LIN {X -0.023,Y -429.187,Z 1281.514,A 0.000,B 0.000,C 90.000,E1 272.465} C_DIS
LIN {X -0.033,Y -422.236,Z 1281.512,A 0.000,B 0.000,C 90.000,E1 272.121} C_DIS
LIN {X -0.038,Y -415.238,Z 1281.510,A 0.000,B 0.000,C 90.000,E1 271.835} C_DIS
LIN {X -0.099,Y -408.071,Z 1281.509,A 0.000,B 0.000,C 90.000,E1 271.604} C_DIS
LIN {X 0.103,Y -401.016,Z 1281.508,A 0.000,B 0.000,C 90.000,E1 271.375} C_DIS
LIN {X 0.112,Y -393.582,Z 1281.507,A 0.000,B 0.000,C 90.000,E1 271.203} C_DIS
LIN {X -0.037,Y -385.526,Z 1281.506,A 0.000,B 0.000,C 90.000,E1 271.088} C_DIS
LIN {X 0.028,Y -376.510,Z 1281.505,A 0.000,B 0.000,C 90.000,E1 270.974} C_DIS
LIN {X -0.122,Y -364.751,Z 1281.505,A 0.000,B 0.000,C 90.000,E1 270.917} C_DIS
LIN {X -0.176,Y -360.433,Z 1281.505,A 0.000,B 0.000,C 90.000,E1 270.917} C_DIS
LIN {X 0.065,Y -181.483,Z 1281.505,A 0.000,B 0.000,C 90.000,E1 270.859} C_DIS
LIN {X 0.085,Y -181.533,Z 1281.499,A 0.000,B 0.000,C 90.000,E1 269.828} C_DIS
LIN {X 0.028,Y -180.907,Z 1281.475,A 0.000,B 0.000,C 90.000,E1 265.469} C_DIS
LIN {X -0.095,Y -180.741,Z 1281.470,A 0.000,B 0.000,C 90.000,E1 264.666} C_DIS
LIN {X 0.006,Y -178.831,Z 1281.442,A 0.000,B 0.000,C 90.000,E1 259.567} C_DIS
LIN {X 0.040,Y -175.875,Z 1281.414,A 0.000,B 0.000,C 90.000,E1 254.464} C_DIS
LIN {X -0.084,Y -173.849,Z 1281.400,A 0.000,B 0.000,C 90.000,E1 251.945} C_DIS
LIN {X 0.070,Y -171.518,Z 1281.380,A 0.000,B 0.000,C 90.000,E1 248.465} C_DIS
LIN {X 0.056,Y -167.744,Z 1281.357,A 0.000,B 0.000,C 90.000,E1 244.152} C_DIS
LIN {X 0.072,Y -166.446,Z 1281.347,A 0.000,B 0.000,C 90.000,E1 242.410} C_DIS
LIN {X -0.016,Y -163.163,Z 1281.328,A 0.000,B 0.000,C 90.000,E1 238.948} C_DIS
LIN {X 0.034,Y -161.121,Z 1281.313,A 0.000,B 0.000,C 90.000,E1 236.294} C_DIS
LIN {X -0.063,Y -157.144,Z 1281.288,A 0.000,B 0.000,C 90.000,E1 231.904} C_DIS
LIN {X -0.040,Y -155.877,Z 1281.278,A 0.000,B 0.000,C 90.000,E1 230.114} C_DIS
LIN {X -0.081,Y -152.127,Z 1281.253,A 0.000,B 0.000,C 90.000,E1 225.648} C_DIS
LIN {X -0.060,Y -150.377,Z 1281.238,A 0.000,B 0.000,C 90.000,E1 222.933} C_DIS
LIN {X -0.035,Y -147.110,Z 1281.213,A 0.000,B 0.000,C 90.000,E1 218.382} C_DIS
LIN {X -0.044,Y -145.676,Z 1281.198,A 0.000,B 0.000,C 90.000,E1 215.644} C_DIS
LIN {X -0.046,Y -143.059,Z 1281.172,A 0.000,B 0.000,C 90.000,E1 211.052} C_DIS
LIN {X 0.012,Y -141.681,Z 1281.152,A 0.000,B 0.000,C 90.000,E1 207.334} C_DIS
LIN {X -0.010,Y -139.457,Z 1281.116,A 0.000,B 0.000,C 90.000,E1 200.844} C_DIS
LIN {X 0.040,Y -139.191,Z 1281.105,A 0.000,B 0.000,C 90.000,E1 198.960} C_DIS
LIN {X 0.064,Y -138.324,Z 1281.054,A 0.000,B 0.000,C 90.000,E1 189.613} C_DIS
LIN {X -0.068,Y -139.455,Z 1281.007,A 0.000,B 0.000,C 90.000,E1 181.260} C_DIS
LIN {X 0.012,Y -141.005,Z 1280.976,A 0.000,B 0.000,C 90.000,E1 175.641} C_DIS
LIN {X -0.039,Y -142.759,Z 1280.955,A 0.000,B 0.000,C 90.000,E1 171.951} C_DIS
LIN {X 0.058,Y -145.164,Z 1280.930,A 0.000,B 0.000,C 90.000,E1 167.297} C_DIS
LIN {X 0.050,Y -147.786,Z 1280.909,A 0.000,B 0.000,C 90.000,E1 163.630} C_DIS
LIN {X -0.012,Y -150.466,Z 1280.889,A 0.000,B 0.000,C 90.000,E1 160.007} C_DIS
LIN {X 0.062,Y -153.918,Z 1280.869,A 0.000,B 0.000,C 90.000,E1 156.357} C_DIS
LIN {X -0.013,Y -157.329,Z 1280.849,A 0.000,B 0.000,C 90.000,E1 152.794} C_DIS
LIN {X 0.071,Y -161.519,Z 1280.829,A 0.000,B 0.000,C 90.000,E1 149.203} C_DIS
LIN {X -0.053,Y -165.718,Z 1280.809,A 0.000,B 0.000,C 90.000,E1 145.722} C_DIS
LIN {X 0.072,Y -170.666,Z 1280.790,A 0.000,B 0.000,C 90.000,E1 142.190} C_DIS
LIN {X -0.015,Y -175.541,Z 1280.771,A 0.000,B 0.000,C 90.000,E1 138.771} C_DIS
LIN {X -0.022,Y -181.160,Z 1280.752,A 0.000,B 0.000,C 90.000,E1 135.364} C_DIS
LIN {X -0.025,Y -186.614,Z 1280.733,A 0.000,B 0.000,C 90.000,E1 132.000} C_DIS
LIN {X 0.046,Y -191.223,Z 1280.719,A 0.000,B 0.000,C 90.000,E1 129.483} C_DIS
LIN {X -0.032,Y -197.039,Z 1280.701,A 0.000,B 0.000,C 90.000,E1 126.217} C_DIS
LIN {X -0.072,Y -199.854,Z 1280.693,A 0.000,B 0.000,C 90.000,E1 124.818} C_DIS
LIN {X -0.149,Y -309.309,Z 1280.693,A 0.000,B 0.000,C 90.000,E1 124.818} C_DIS
LIN {X -0.180,Y -315.387,Z 1280.692,A 0.000,B 0.000,C 90.000,E1 124.612} C_DIS
LIN {X 0.081,Y -318.330,Z 1280.691,A 0.000,B 0.000,C 90.000,E1 124.326} C_DIS
LIN {X 0.009,Y -322.051,Z 1280.688,A 0.000,B 0.000,C 90.000,E1 123.865} C_DIS
LIN {X -0.184,Y -323.801,Z 1280.686,A 0.000,B 0.000,C 90.000,E1 123.579} C_DIS
LIN {X 0.070,Y -325.164,Z 1280.685,A 0.000,B 0.000,C 90.000,E1 123.214} C_DIS
LIN {X 0.002,Y -336.874,Z 1280.667,A 0.000,B 0.000,C 90.000,E1 120.079} C_DIS
LIN {X -0.030,Y -348.823,Z 1280.652,A 0.000,B 0.000,C 90.000,E1 117.308} C_DIS
LIN {X -0.055,Y -362.234,Z 1280.637,A 0.000,B 0.000,C 90.000,E1 114.591} C_DIS
LIN {X 0.061,Y -375.474,Z 1280.623,A 0.000,B 0.000,C 90.000,E1 112.206} C_DIS
LIN {X 0.091,Y -390.050,Z 1280.611,A 0.000,B 0.000,C 90.000,E1 109.885} C_DIS
LIN {X -0.017,Y -406.067,Z 1280.598,A 0.000,B 0.000,C 90.000,E1 107.638} C_DIS
LIN {X 0.015,Y -423.637,Z 1280.586,A 0.000,B 0.000,C 90.000,E1 105.426} C_DIS
LIN {X -0.129,Y -442.844,Z 1280.574,A 0.000,B 0.000,C 90.000,E1 103.300} C_DIS
LIN {X -0.134,Y -462.963,Z 1280.563,A 0.000,B 0.000,C 90.000,E1 101.299} C_DIS
LIN {X -0.203,Y -475.789,Z 1280.556,A 0.000,B 0.000,C 90.000,E1 100.141} C_DIS
LIN {X -0.134,Y -477.907,Z 1280.555,A 0.000,B 0.000,C 90.000,E1 99.905} C_DIS
LIN {X 0.209,Y -479.663,Z 1280.554,A 0.000,B 0.000,C 90.000,E1 99.613} C_DIS
LIN {X 0.077,Y -480.981,Z 1280.552,A 0.000,B 0.000,C 90.000,E1 99.378} C_DIS
LIN {X 0.233,Y -482.621,Z 1280.549,A 0.000,B 0.000,C 90.000,E1 98.859} C_DIS
LIN {X -0.078,Y -483.190,Z 1280.547,A 0.000,B 0.000,C 90.000,E1 98.398} C_DIS
LIN {X 0.166,Y -482.782,Z 1280.544,A 0.000,B 0.000,C 90.000,E1 97.871} C_DIS
LIN {X -0.133,Y -481.337,Z 1280.541,A 0.000,B 0.000,C 90.000,E1 97.409} C_DIS
LIN {X 0.164,Y -480.150,Z 1280.540,A 0.000,B 0.000,C 90.000,E1 97.125} C_DIS
LIN {X 0.043,Y -478.567,Z 1280.538,A 0.000,B 0.000,C 90.000,E1 96.891} C_DIS
LIN {X 0.044,Y -463.775,Z 1280.527,A 0.000,B 0.000,C 90.000,E1 94.878} C_DIS
LIN {X 0.139,Y -446.409,Z 1280.513,A 0.000,B 0.000,C 90.000,E1 92.293} C_DIS
LIN {X -0.012,Y -431.889,Z 1280.500,A 0.000,B 0.000,C 90.000,E1 89.943} C_DIS
LIN {X 0.013,Y -417.151,Z 1280.485,A 0.000,B 0.000,C 90.000,E1 87.249} C_DIS
LIN {X -0.060,Y -405.581,Z 1280.473,A 0.000,B 0.000,C 90.000,E1 85.065} C_DIS
LIN {X -0.059,Y -396.894,Z 1280.463,A 0.000,B 0.000,C 90.000,E1 83.394} C_DIS
LIN {X -0.166,Y -386.549,Z 1280.452,A 0.000,B 0.000,C 90.000,E1 81.432} C_DIS
LIN {X -0.022,Y -377.434,Z 1280.443,A 0.000,B 0.000,C 90.000,E1 79.690} C_DIS
LIN {X 0.022,Y -367.963,Z 1280.433,A 0.000,B 0.000,C 90.000,E1 77.937} C_DIS
LIN {X -0.027,Y -358.150,Z 1280.423,A 0.000,B 0.000,C 90.000,E1 76.172} C_DIS
LIN {X 0.097,Y -346.573,Z 1280.411,A 0.000,B 0.000,C 90.000,E1 74.047} C_DIS
LIN {X -0.162,Y -335.085,Z 1280.400,A 0.000,B 0.000,C 90.000,E1 71.945} C_DIS
LIN {X 0.088,Y -320.715,Z 1280.384,A 0.000,B 0.000,C 90.000,E1 69.082} C_DIS
LIN {X 0.105,Y -304.373,Z 1280.364,A 0.000,B 0.000,C 90.000,E1 65.537} C_DIS
LIN {X -0.024,Y -293.664,Z 1280.349,A 0.000,B 0.000,C 90.000,E1 62.922} C_DIS
LIN {X 0.112,Y -284.252,Z 1280.335,A 0.000,B 0.000,C 90.000,E1 60.205} C_DIS
LIN {X -0.136,Y -273.724,Z 1280.316,A 0.000,B 0.000,C 90.000,E1 56.834} C_DIS
LIN {X -0.077,Y -264.169,Z 1280.296,A 0.000,B 0.000,C 90.000,E1 53.336} C_DIS
LIN {X 0.018,Y -256.937,Z 1280.281,A 0.000,B 0.000,C 90.000,E1 50.481} C_DIS
LIN {X -0.105,Y -249.955,Z 1280.265,A 0.000,B 0.000,C 90.000,E1 47.634} C_DIS
LIN {X 0.057,Y -241.694,Z 1280.244,A 0.000,B 0.000,C 90.000,E1 43.947} C_DIS
LIN {X -0.012,Y -233.958,Z 1280.224,A 0.000,B 0.000,C 90.000,E1 40.253} C_DIS
LIN {X -0.080,Y -227.073,Z 1280.203,A 0.000,B 0.000,C 90.000,E1 36.503} C_DIS
LIN {X -0.041,Y -220.916,Z 1280.182,A 0.000,B 0.000,C 90.000,E1 32.673} C_DIS
LIN {X -0.103,Y -215.433,Z 1280.160,A 0.000,B 0.000,C 90.000,E1 28.821} C_DIS
LIN {X -0.068,Y -210.589,Z 1280.138,A 0.000,B 0.000,C 90.000,E1 24.899} C_DIS
LIN {X 0.046,Y -205.645,Z 1280.112,A 0.000,B 0.000,C 90.000,E1 20.120} C_DIS
LIN {X 0.072,Y -201.484,Z 1280.085,A 0.000,B 0.000,C 90.000,E1 15.315} C_DIS
LIN {X 0.062,Y -197.828,Z 1280.054,A 0.000,B 0.000,C 90.000,E1 9.670} C_DIS
LIN {X 0.062,Y -195.327,Z 1280.013,A 0.000,B 0.000,C 90.000,E1 2.350} C_DIS
LIN {X 0.014,Y -196.745,Z 1279.957,A 0.000,B 0.000,C 90.000,E1 352.186} C_DIS
LIN {X -0.045,Y -200.083,Z 1279.925,A 0.000,B 0.000,C 90.000,E1 346.520} C_DIS
LIN {X -0.067,Y -204.142,Z 1279.898,A 0.000,B 0.000,C 90.000,E1 341.692} C_DIS
LIN {X 0.045,Y -208.261,Z 1279.876,A 0.000,B 0.000,C 90.000,E1 337.667} C_DIS
LIN {X 0.020,Y -213.164,Z 1279.854,A 0.000,B 0.000,C 90.000,E1 333.717} C_DIS
LIN {X 0.055,Y -218.767,Z 1279.832,A 0.000,B 0.000,C 90.000,E1 329.793} C_DIS
LIN {X 0.047,Y -225.145,Z 1279.811,A 0.000,B 0.000,C 90.000,E1 325.928} C_DIS
LIN {X 0.065,Y -232.457,Z 1279.790,A 0.000,B 0.000,C 90.000,E1 322.110} C_DIS
LIN {X 0.016,Y -240.603,Z 1279.769,A 0.000,B 0.000,C 90.000,E1 318.366} C_DIS
LIN {X 0.016,Y -248.933,Z 1279.750,A 0.000,B 0.000,C 90.000,E1 315.040} C_DIS
LIN {X 0.065,Y -257.259,Z 1279.734,A 0.000,B 0.000,C 90.000,E1 312.123} C_DIS
LIN {X -0.089,Y -264.405,Z 1279.722,A 0.000,B 0.000,C 90.000,E1 310.011} C_DIS
LIN {X 0.019,Y -271.052,Z 1279.712,A 0.000,B 0.000,C 90.000,E1 308.222} C_DIS
LIN {X -0.001,Y -279.977,Z 1279.701,A 0.000,B 0.000,C 90.000,E1 306.137} C_DIS
LIN {X 0.059,Y -289.953,Z 1279.689,A 0.000,B 0.000,C 90.000,E1 304.072} C_DIS
LIN {X -0.085,Y -301.013,Z 1279.678,A 0.000,B 0.000,C 90.000,E1 302.084} C_DIS
LIN {X 0.038,Y -311.291,Z 1279.669,A 0.000,B 0.000,C 90.000,E1 300.413} C_DIS
LIN {X 0.059,Y -327.603,Z 1279.656,A 0.000,B 0.000,C 90.000,E1 298.153} C_DIS
LIN {X -0.025,Y -347.797,Z 1279.643,A 0.000,B 0.000,C 90.000,E1 295.668} C_DIS
LIN {X 0.113,Y -360.704,Z 1279.634,A 0.000,B 0.000,C 90.000,E1 294.155} C_DIS
LIN {X -0.040,Y -373.638,Z 1279.626,A 0.000,B 0.000,C 90.000,E1 292.695} C_DIS
LIN {X -0.144,Y -386.003,Z 1279.618,A 0.000,B 0.000,C 90.000,E1 291.280} C_DIS
LIN {X 0.233,Y -410.888,Z 1279.603,A 0.000,B 0.000,C 90.000,E1 288.417} C_DIS
LIN {X 0.117,Y -420.946,Z 1279.596,A 0.000,B 0.000,C 90.000,E1 287.347} C_DIS
LIN {X 0.132,Y -430.448,Z 1279.590,A 0.000,B 0.000,C 90.000,E1 286.260} C_DIS
LIN {X -0.066,Y -437.039,Z 1279.586,A 0.000,B 0.000,C 90.000,E1 285.481} C_DIS
LIN {X 0.109,Y -443.024,Z 1279.582,A 0.000,B 0.000,C 90.000,E1 284.662} C_DIS
LIN {X 0.017,Y -448.346,Z 1279.577,A 0.000,B 0.000,C 90.000,E1 283.883} C_DIS
LIN {X -0.136,Y -452.992,Z 1279.573,A 0.000,B 0.000,C 90.000,E1 283.119} C_DIS
LIN {X 0.193,Y -456.947,Z 1279.568,A 0.000,B 0.000,C 90.000,E1 282.299} C_DIS
LIN {X -0.162,Y -459.237,Z 1279.566,A 0.000,B 0.000,C 90.000,E1 281.827} C_DIS
LIN {X -0.056,Y -461.228,Z 1279.563,A 0.000,B 0.000,C 90.000,E1 281.299} C_DIS
LIN {X -0.031,Y -462.946,Z 1279.560,A 0.000,B 0.000,C 90.000,E1 280.782} C_DIS
LIN {X 0.094,Y -464.342,Z 1279.557,A 0.000,B 0.000,C 90.000,E1 280.254} C_DIS
LIN {X 0.226,Y -465.390,Z 1279.554,A 0.000,B 0.000,C 90.000,E1 279.726} C_DIS
LIN {X -0.171,Y -466.115,Z 1279.551,A 0.000,B 0.000,C 90.000,E1 279.265} C_DIS
LIN {X -0.099,Y -466.471,Z 1279.548,A 0.000,B 0.000,C 90.000,E1 278.746} C_DIS
LIN {X 0.046,Y -466.382,Z 1279.546,A 0.000,B 0.000,C 90.000,E1 278.219} C_DIS
LIN {X 0.125,Y -465.867,Z 1279.543,A 0.000,B 0.000,C 90.000,E1 277.701} C_DIS
LIN {X 0.205,Y -464.875,Z 1279.540,A 0.000,B 0.000,C 90.000,E1 277.182} C_DIS
LIN {X -0.178,Y -463.420,Z 1279.537,A 0.000,B 0.000,C 90.000,E1 276.720} C_DIS
LIN {X -0.105,Y -461.545,Z 1279.534,A 0.000,B 0.000,C 90.000,E1 276.201} C_DIS
LIN {X 0.231,Y -458.114,Z 1279.530,A 0.000,B 0.000,C 90.000,E1 275.391} C_DIS
LIN {X -0.227,Y -455.355,Z 1279.527,A 0.000,B 0.000,C 90.000,E1 274.935} C_DIS
LIN {X -0.203,Y -452.069,Z 1279.524,A 0.000,B 0.000,C 90.000,E1 274.416} C_DIS
LIN {X -0.198,Y -447.836,Z 1279.521,A 0.000,B 0.000,C 90.000,E1 273.898} C_DIS
LIN {X 0.007,Y -445.358,Z 1279.520,A 0.000,B 0.000,C 90.000,E1 273.612} C_DIS
LIN {X -0.003,Y -439.433,Z 1279.517,A 0.000,B 0.000,C 90.000,E1 273.094} C_DIS
LIN {X 0.067,Y -432.981,Z 1279.515,A 0.000,B 0.000,C 90.000,E1 272.636} C_DIS
LIN {X 0.187,Y -426.045,Z 1279.513,A 0.000,B 0.000,C 90.000,E1 272.236} C_DIS
LIN {X -0.035,Y -419.065,Z 1279.511,A 0.000,B 0.000,C 90.000,E1 271.949} C_DIS
LIN {X 0.193,Y -412.131,Z 1279.509,A 0.000,B 0.000,C 90.000,E1 271.661} C_DIS
LIN {X -0.145,Y -405.059,Z 1279.508,A 0.000,B 0.000,C 90.000,E1 271.489} C_DIS
LIN {X 0.141,Y -397.896,Z 1279.507,A 0.000,B 0.000,C 90.000,E1 271.260} C_DIS
LIN {X -0.184,Y -389.490,Z 1279.506,A 0.000,B 0.000,C 90.000,E1 271.146} C_DIS
LIN {X 0.174,Y -381.137,Z 1279.506,A 0.000,B 0.000,C 90.000,E1 270.974} C_DIS
LIN {X -0.073,Y -370.345,Z 1279.505,A 0.000,B 0.000,C 90.000,E1 270.917} C_DIS
LIN {X 0.010,Y -359.049,Z 1279.505,A 0.000,B 0.000,C 90.000,E1 270.859} C_DIS
LIN {X -0.023,Y -181.490,Z 1279.505,A 0.000,B 0.000,C 90.000,E1 270.859} C_DIS
LIN {X -0.002,Y -181.525,Z 1279.499,A 0.000,B 0.000,C 90.000,E1 269.828} C_DIS
LIN {X -0.059,Y -180.907,Z 1279.475,A 0.000,B 0.000,C 90.000,E1 265.469} C_DIS
LIN {X -0.003,Y -180.728,Z 1279.470,A 0.000,B 0.000,C 90.000,E1 264.609} C_DIS
LIN {X 0.095,Y -178.817,Z 1279.442,A 0.000,B 0.000,C 90.000,E1 259.511} C_DIS
LIN {X 0.001,Y -175.861,Z 1279.414,A 0.000,B 0.000,C 90.000,E1 254.448} C_DIS
LIN {X 0.050,Y -173.827,Z 1279.399,A 0.000,B 0.000,C 90.000,E1 251.873} C_DIS
LIN {X -0.014,Y -171.495,Z 1279.380,A 0.000,B 0.000,C 90.000,E1 248.465} C_DIS
LIN {X -0.028,Y -167.724,Z 1279.356,A 0.000,B 0.000,C 90.000,E1 244.152} C_DIS
LIN {X -0.012,Y -166.417,Z 1279.347,A 0.000,B 0.000,C 90.000,E1 242.410} C_DIS
LIN {X -0.013,Y -163.140,Z 1279.327,A 0.000,B 0.000,C 90.000,E1 238.918} C_DIS
LIN {X -0.048,Y -161.093,Z 1279.313,A 0.000,B 0.000,C 90.000,E1 236.294} C_DIS
LIN {X -0.064,Y -157.822,Z 1279.293,A 0.000,B 0.000,C 90.000,E1 232.763} C_DIS
LIN {X 0.000,Y -155.856,Z 1279.278,A 0.000,B 0.000,C 90.000,E1 230.070} C_DIS
LIN {X 0.055,Y -152.105,Z 1279.253,A 0.000,B 0.000,C 90.000,E1 225.567} C_DIS
LIN {X 0.074,Y -150.356,Z 1279.238,A 0.000,B 0.000,C 90.000,E1 222.852} C_DIS
LIN {X 0.002,Y -147.092,Z 1279.213,A 0.000,B 0.000,C 90.000,E1 218.338} C_DIS
LIN {X -0.003,Y -145.663,Z 1279.198,A 0.000,B 0.000,C 90.000,E1 215.598} C_DIS
LIN {X 0.001,Y -143.045,Z 1279.172,A 0.000,B 0.000,C 90.000,E1 211.003} C_DIS
LIN {X 0.001,Y -141.669,Z 1279.152,A 0.000,B 0.000,C 90.000,E1 207.308} C_DIS
LIN {X 0.046,Y -139.451,Z 1279.116,A 0.000,B 0.000,C 90.000,E1 200.791} C_DIS
LIN {X -0.034,Y -139.186,Z 1279.105,A 0.000,B 0.000,C 90.000,E1 198.960} C_DIS
LIN {X -0.011,Y -138.321,Z 1279.053,A 0.000,B 0.000,C 90.000,E1 189.613} C_DIS
LIN {X -0.003,Y -139.461,Z 1279.007,A 0.000,B 0.000,C 90.000,E1 181.203} C_DIS
LIN {X -0.064,Y -141.018,Z 1278.976,A 0.000,B 0.000,C 90.000,E1 175.641} C_DIS
LIN {X 0.027,Y -142.772,Z 1278.955,A 0.000,B 0.000,C 90.000,E1 171.894} C_DIS
LIN {X 0.013,Y -145.184,Z 1278.929,A 0.000,B 0.000,C 90.000,E1 167.285} C_DIS
LIN {X 0.015,Y -147.805,Z 1278.909,A 0.000,B 0.000,C 90.000,E1 163.614} C_DIS
LIN {X -0.091,Y -150.491,Z 1278.889,A 0.000,B 0.000,C 90.000,E1 160.007} C_DIS
LIN {X -0.018,Y -153.949,Z 1278.869,A 0.000,B 0.000,C 90.000,E1 156.357} C_DIS
LIN {X 0.045,Y -157.359,Z 1278.849,A 0.000,B 0.000,C 90.000,E1 152.743} C_DIS
LIN {X -0.011,Y -161.557,Z 1278.829,A 0.000,B 0.000,C 90.000,E1 149.203} C_DIS
LIN {X 0.000,Y -165.755,Z 1278.809,A 0.000,B 0.000,C 90.000,E1 145.674} C_DIS
LIN {X -0.013,Y -170.710,Z 1278.790,A 0.000,B 0.000,C 90.000,E1 142.190} C_DIS
LIN {X 0.031,Y -175.583,Z 1278.771,A 0.000,B 0.000,C 90.000,E1 138.728} C_DIS
LIN {X 0.018,Y -181.201,Z 1278.752,A 0.000,B 0.000,C 90.000,E1 135.324} C_DIS
LIN {X 0.011,Y -186.663,Z 1278.733,A 0.000,B 0.000,C 90.000,E1 131.962} C_DIS
LIN {X -0.045,Y -191.268,Z 1278.719,A 0.000,B 0.000,C 90.000,E1 129.483} C_DIS
LIN {X 0.035,Y -197.090,Z 1278.701,A 0.000,B 0.000,C 90.000,E1 126.171} C_DIS
LIN {X -0.115,Y -199.881,Z 1278.693,A 0.000,B 0.000,C 90.000,E1 124.818} C_DIS
LIN {X 0.039,Y -309.317,Z 1278.693,A 0.000,B 0.000,C 90.000,E1 124.771} C_DIS
LIN {X 0.104,Y -310.853,Z 1278.693,A 0.000,B 0.000,C 90.000,E1 124.739} C_DIS
LIN {X 0.112,Y -315.626,Z 1278.692,A 0.000,B 0.000,C 90.000,E1 124.532} C_DIS
LIN {X 0.034,Y -318.780,Z 1278.690,A 0.000,B 0.000,C 90.000,E1 124.278} C_DIS
LIN {X 0.040,Y -322.447,Z 1278.688,A 0.000,B 0.000,C 90.000,E1 123.785} C_DIS
LIN {X -0.153,Y -324.111,Z 1278.686,A 0.000,B 0.000,C 90.000,E1 123.499} C_DIS
LIN {X 0.021,Y -326.513,Z 1278.682,A 0.000,B 0.000,C 90.000,E1 122.832} C_DIS
LIN {X 0.038,Y -337.143,Z 1278.667,A 0.000,B 0.000,C 90.000,E1 120.001} C_DIS
LIN {X -0.152,Y -349.128,Z 1278.651,A 0.000,B 0.000,C 90.000,E1 117.257} C_DIS
LIN {X -0.015,Y -362.578,Z 1278.636,A 0.000,B 0.000,C 90.000,E1 114.515} C_DIS
LIN {X -0.038,Y -375.854,Z 1278.623,A 0.000,B 0.000,C 90.000,E1 112.153} C_DIS
LIN {X 0.136,Y -390.471,Z 1278.610,A 0.000,B 0.000,C 90.000,E1 109.812} C_DIS
LIN {X -0.092,Y -406.531,Z 1278.598,A 0.000,B 0.000,C 90.000,E1 107.583} C_DIS
LIN {X -0.047,Y -424.147,Z 1278.585,A 0.000,B 0.000,C 90.000,E1 105.371} C_DIS
LIN {X -0.170,Y -443.398,Z 1278.573,A 0.000,B 0.000,C 90.000,E1 103.244} C_DIS
LIN {X -0.135,Y -463.534,Z 1278.562,A 0.000,B 0.000,C 90.000,E1 101.243} C_DIS
LIN {X -0.095,Y -476.300,Z 1278.556,A 0.000,B 0.000,C 90.000,E1 100.074} C_DIS
LIN {X -0.103,Y -478.251,Z 1278.555,A 0.000,B 0.000,C 90.000,E1 99.849} C_DIS
LIN {X -0.233,Y -479.885,Z 1278.553,A 0.000,B 0.000,C 90.000,E1 99.613} C_DIS
LIN {X 0.111,Y -481.109,Z 1278.552,A 0.000,B 0.000,C 90.000,E1 99.321} C_DIS
LIN {X -0.208,Y -482.606,Z 1278.549,A 0.000,B 0.000,C 90.000,E1 98.859} C_DIS
LIN {X -0.041,Y -483.053,Z 1278.546,A 0.000,B 0.000,C 90.000,E1 98.341} C_DIS
LIN {X 0.203,Y -482.525,Z 1278.544,A 0.000,B 0.000,C 90.000,E1 97.814} C_DIS
LIN {X -0.096,Y -480.940,Z 1278.541,A 0.000,B 0.000,C 90.000,E1 97.352} C_DIS
LIN {X 0.200,Y -479.664,Z 1278.539,A 0.000,B 0.000,C 90.000,E1 97.068} C_DIS
LIN {X -0.105,Y -476.050,Z 1278.537,A 0.000,B 0.000,C 90.000,E1 96.606} C_DIS
LIN {X 0.187,Y -456.152,Z 1278.521,A 0.000,B 0.000,C 90.000,E1 93.784} C_DIS
LIN {X 0.202,Y -437.608,Z 1278.505,A 0.000,B 0.000,C 90.000,E1 90.917} C_DIS
LIN {X 0.085,Y -420.993,Z 1278.489,A 0.000,B 0.000,C 90.000,E1 87.993} C_DIS
LIN {X -0.032,Y -410.826,Z 1278.478,A 0.000,B 0.000,C 90.000,E1 86.102} C_DIS
LIN {X 0.104,Y -400.755,Z 1278.468,A 0.000,B 0.000,C 90.000,E1 84.147} C_DIS
LIN {X 0.059,Y -391.959,Z 1278.458,A 0.000,B 0.000,C 90.000,E1 82.470} C_DIS
LIN {X -0.135,Y -383.032,Z 1278.449,A 0.000,B 0.000,C 90.000,E1 80.792} C_DIS
LIN {X -0.055,Y -373.799,Z 1278.439,A 0.000,B 0.000,C 90.000,E1 79.050} C_DIS
LIN {X 0.001,Y -364.189,Z 1278.429,A 0.000,B 0.000,C 90.000,E1 77.285} C_DIS
LIN {X -0.111,Y -354.302,Z 1278.419,A 0.000,B 0.000,C 90.000,E1 75.519} C_DIS
LIN {X 0.030,Y -342.736,Z 1278.408,A 0.000,B 0.000,C 90.000,E1 73.378} C_DIS
LIN {X 0.018,Y -331.311,Z 1278.396,A 0.000,B 0.000,C 90.000,E1 71.221} C_DIS
LIN {X -0.142,Y -317.169,Z 1278.380,A 0.000,B 0.000,C 90.000,E1 68.411} C_DIS
LIN {X -0.010,Y -302.578,Z 1278.362,A 0.000,B 0.000,C 90.000,E1 65.153} C_DIS
LIN {X 0.089,Y -293.315,Z 1278.349,A 0.000,B 0.000,C 90.000,E1 62.820} C_DIS
LIN {X 0.067,Y -282.815,Z 1278.332,A 0.000,B 0.000,C 90.000,E1 59.793} C_DIS
LIN {X 0.105,Y -271.391,Z 1278.311,A 0.000,B 0.000,C 90.000,E1 56.008} C_DIS
LIN {X -0.132,Y -261.948,Z 1278.292,A 0.000,B 0.000,C 90.000,E1 52.557} C_DIS
LIN {X 0.067,Y -254.786,Z 1278.276,A 0.000,B 0.000,C 90.000,E1 49.666} C_DIS
LIN {X 0.051,Y -247.863,Z 1278.260,A 0.000,B 0.000,C 90.000,E1 46.782} C_DIS
LIN {X -0.031,Y -239.732,Z 1278.240,A 0.000,B 0.000,C 90.000,E1 43.137} C_DIS
LIN {X 0.011,Y -232.146,Z 1278.219,A 0.000,B 0.000,C 90.000,E1 39.402} C_DIS
LIN {X 0.103,Y -225.408,Z 1278.198,A 0.000,B 0.000,C 90.000,E1 35.598} C_DIS
LIN {X -0.033,Y -219.368,Z 1278.177,A 0.000,B 0.000,C 90.000,E1 31.799} C_DIS
LIN {X 0.044,Y -213.971,Z 1278.155,A 0.000,B 0.000,C 90.000,E1 27.897} C_DIS
LIN {X -0.044,Y -208.360,Z 1278.129,A 0.000,B 0.000,C 90.000,E1 23.206} C_DIS
LIN {X 0.030,Y -204.388,Z 1278.107,A 0.000,B 0.000,C 90.000,E1 19.214} C_DIS
LIN {X 0.006,Y -200.386,Z 1278.080,A 0.000,B 0.000,C 90.000,E1 14.411} C_DIS
LIN {X 0.021,Y -197.007,Z 1278.049,A 0.000,B 0.000,C 90.000,E1 8.746} C_DIS
LIN {X 0.000,Y -194.842,Z 1278.000,A 0.000,B 0.000,C 90.000,E1 360.000} C_DIS
LIN {X -0.015,Y -196.955,Z 1277.952,A 0.000,B 0.000,C 90.000,E1 351.376} C_DIS
LIN {X -0.025,Y -200.598,Z 1277.921,A 0.000,B 0.000,C 90.000,E1 345.700} C_DIS
LIN {X 0.022,Y -204.837,Z 1277.894,A 0.000,B 0.000,C 90.000,E1 340.859} C_DIS
LIN {X 0.029,Y -209.163,Z 1277.872,A 0.000,B 0.000,C 90.000,E1 336.869} C_DIS
LIN {X 0.021,Y -214.204,Z 1277.850,A 0.000,B 0.000,C 90.000,E1 332.922} C_DIS
LIN {X 0.097,Y -219.966,Z 1277.828,A 0.000,B 0.000,C 90.000,E1 328.997} C_DIS
LIN {X -0.066,Y -226.542,Z 1277.807,A 0.000,B 0.000,C 90.000,E1 325.182} C_DIS
LIN {X -0.057,Y -234.041,Z 1277.785,A 0.000,B 0.000,C 90.000,E1 321.376} C_DIS
LIN {X -0.065,Y -242.379,Z 1277.765,A 0.000,B 0.000,C 90.000,E1 317.634} C_DIS
LIN {X -0.031,Y -251.916,Z 1277.744,A 0.000,B 0.000,C 90.000,E1 313.947} C_DIS
LIN {X 0.095,Y -259.526,Z 1277.730,A 0.000,B 0.000,C 90.000,E1 311.391} C_DIS
LIN {X -0.010,Y -266.950,Z 1277.718,A 0.000,B 0.000,C 90.000,E1 309.277} C_DIS
LIN {X -0.027,Y -273.884,Z 1277.708,A 0.000,B 0.000,C 90.000,E1 307.523} C_DIS
LIN {X 0.011,Y -283.153,Z 1277.697,A 0.000,B 0.000,C 90.000,E1 305.438} C_DIS
LIN {X 0.137,Y -293.485,Z 1277.686,A 0.000,B 0.000,C 90.000,E1 303.372} C_DIS
LIN {X 0.044,Y -302.915,Z 1277.676,A 0.000,B 0.000,C 90.000,E1 301.720} C_DIS
LIN {X -0.008,Y -311.200,Z 1277.669,A 0.000,B 0.000,C 90.000,E1 300.413} C_DIS
LIN {X 0.008,Y -327.553,Z 1277.656,A 0.000,B 0.000,C 90.000,E1 298.153} C_DIS
LIN {X -0.064,Y -347.717,Z 1277.643,A 0.000,B 0.000,C 90.000,E1 295.668} C_DIS
LIN {X 0.060,Y -360.651,Z 1277.634,A 0.000,B 0.000,C 90.000,E1 294.155} C_DIS
LIN {X -0.094,Y -373.586,Z 1277.626,A 0.000,B 0.000,C 90.000,E1 292.695} C_DIS
LIN {X -0.016,Y -386.211,Z 1277.618,A 0.000,B 0.000,C 90.000,E1 291.227} C_DIS
LIN {X 0.208,Y -410.901,Z 1277.602,A 0.000,B 0.000,C 90.000,E1 288.417} C_DIS
LIN {X 0.109,Y -420.945,Z 1277.596,A 0.000,B 0.000,C 90.000,E1 287.347} C_DIS
LIN {X 0.132,Y -430.438,Z 1277.590,A 0.000,B 0.000,C 90.000,E1 286.260} C_DIS
LIN {X -0.066,Y -437.049,Z 1277.586,A 0.000,B 0.000,C 90.000,E1 285.481} C_DIS
LIN {X 0.108,Y -443.037,Z 1277.582,A 0.000,B 0.000,C 90.000,E1 284.662} C_DIS
LIN {X 0.015,Y -448.361,Z 1277.577,A 0.000,B 0.000,C 90.000,E1 283.883} C_DIS
LIN {X -0.137,Y -453.036,Z 1277.573,A 0.000,B 0.000,C 90.000,E1 283.119} C_DIS
LIN {X 0.192,Y -456.997,Z 1277.568,A 0.000,B 0.000,C 90.000,E1 282.299} C_DIS
LIN {X -0.162,Y -459.281,Z 1277.566,A 0.000,B 0.000,C 90.000,E1 281.827} C_DIS
LIN {X -0.056,Y -461.252,Z 1277.563,A 0.000,B 0.000,C 90.000,E1 281.299} C_DIS
LIN {X -0.031,Y -462.980,Z 1277.560,A 0.000,B 0.000,C 90.000,E1 280.782} C_DIS
LIN {X 0.094,Y -464.363,Z 1277.557,A 0.000,B 0.000,C 90.000,E1 280.254} C_DIS
LIN {X 0.227,Y -465.437,Z 1277.554,A 0.000,B 0.000,C 90.000,E1 279.726} C_DIS
LIN {X -0.170,Y -466.189,Z 1277.551,A 0.000,B 0.000,C 90.000,E1 279.265} C_DIS
LIN {X -0.099,Y -466.527,Z 1277.548,A 0.000,B 0.000,C 90.000,E1 278.746} C_DIS
LIN {X 0.047,Y -466.474,Z 1277.546,A 0.000,B 0.000,C 90.000,E1 278.219} C_DIS
LIN {X 0.127,Y -465.968,Z 1277.543,A 0.000,B 0.000,C 90.000,E1 277.701} C_DIS
LIN {X 0.207,Y -465.020,Z 1277.540,A 0.000,B 0.000,C 90.000,E1 277.182} C_DIS
LIN {X -0.176,Y -463.585,Z 1277.537,A 0.000,B 0.000,C 90.000,E1 276.720} C_DIS
LIN {X -0.102,Y -461.777,Z 1277.534,A 0.000,B 0.000,C 90.000,E1 276.201} C_DIS
LIN {X 0.236,Y -458.372,Z 1277.530,A 0.000,B 0.000,C 90.000,E1 275.391} C_DIS
LIN {X -0.222,Y -455.723,Z 1277.527,A 0.000,B 0.000,C 90.000,E1 274.935} C_DIS
LIN {X -0.195,Y -452.442,Z 1277.524,A 0.000,B 0.000,C 90.000,E1 274.416} C_DIS
LIN {X 0.022,Y -450.550,Z 1277.523,A 0.000,B 0.000,C 90.000,E1 274.131} C_DIS
LIN {X 0.018,Y -445.892,Z 1277.520,A 0.000,B 0.000,C 90.000,E1 273.612} C_DIS
LIN {X 0.211,Y -443.122,Z 1277.519,A 0.000,B 0.000,C 90.000,E1 273.326} C_DIS
LIN {X 0.022,Y -436.981,Z 1277.516,A 0.000,B 0.000,C 90.000,E1 272.865} C_DIS
LIN {X -0.084,Y -430.454,Z 1277.514,A 0.000,B 0.000,C 90.000,E1 272.465} C_DIS
LIN {X -0.113,Y -423.609,Z 1277.512,A 0.000,B 0.000,C 90.000,E1 272.121} C_DIS
LIN {X -0.141,Y -416.630,Z 1277.510,A 0.000,B 0.000,C 90.000,E1 271.835} C_DIS
LIN {X 0.166,Y -409.380,Z 1277.509,A 0.000,B 0.000,C 90.000,E1 271.547} C_DIS
LIN {X 0.050,Y -398.493,Z 1277.507,A 0.000,B 0.000,C 90.000,E1 271.260} C_DIS
LIN {X 0.094,Y -390.110,Z 1277.506,A 0.000,B 0.000,C 90.000,E1 271.088} C_DIS
LIN {X 0.033,Y -381.513,Z 1277.505,A 0.000,B 0.000,C 90.000,E1 270.974} C_DIS
LIN {X 0.162,Y -371.031,Z 1277.505,A 0.000,B 0.000,C 90.000,E1 270.859} C_DIS
LIN {X -0.127,Y -362.447,Z 1277.505,A 0.000,B 0.000,C 90.000,E1 270.859} C_DIS
LIN {X 0.089,Y -181.495,Z 1277.505,A 0.000,B 0.000,C 90.000,E1 270.802} C_DIS
LIN {X -0.072,Y -181.519,Z 1277.499,A 0.000,B 0.000,C 90.000,E1 269.828} C_DIS
LIN {X 0.051,Y -180.907,Z 1277.475,A 0.000,B 0.000,C 90.000,E1 265.412} C_DIS
LIN {X -0.072,Y -180.717,Z 1277.470,A 0.000,B 0.000,C 90.000,E1 264.609} C_DIS
LIN {X 0.026,Y -178.805,Z 1277.442,A 0.000,B 0.000,C 90.000,E1 259.511} C_DIS
LIN {X -0.068,Y -175.850,Z 1277.413,A 0.000,B 0.000,C 90.000,E1 254.448} C_DIS
LIN {X -0.101,Y -172.586,Z 1277.390,A 0.000,B 0.000,C 90.000,E1 250.188} C_DIS
LIN {X 0.077,Y -171.476,Z 1277.380,A 0.000,B 0.000,C 90.000,E1 248.411} C_DIS
LIN {X -0.094,Y -167.707,Z 1277.356,A 0.000,B 0.000,C 90.000,E1 244.152} C_DIS
LIN {X 0.070,Y -166.394,Z 1277.347,A 0.000,B 0.000,C 90.000,E1 242.359} C_DIS
LIN {X 0.061,Y -163.121,Z 1277.327,A 0.000,B 0.000,C 90.000,E1 238.869} C_DIS
LIN {X 0.022,Y -161.070,Z 1277.313,A 0.000,B 0.000,C 90.000,E1 236.246} C_DIS
LIN {X -0.002,Y -157.802,Z 1277.293,A 0.000,B 0.000,C 90.000,E1 232.718} C_DIS
LIN {X -0.063,Y -155.838,Z 1277.278,A 0.000,B 0.000,C 90.000,E1 230.070} C_DIS
LIN {X -0.007,Y -152.089,Z 1277.253,A 0.000,B 0.000,C 90.000,E1 225.567} C_DIS
LIN {X 0.011,Y -150.339,Z 1277.238,A 0.000,B 0.000,C 90.000,E1 222.852} C_DIS
LIN {X 0.032,Y -147.078,Z 1277.213,A 0.000,B 0.000,C 90.000,E1 218.302} C_DIS
LIN {X -0.063,Y -145.652,Z 1277.198,A 0.000,B 0.000,C 90.000,E1 215.598} C_DIS
LIN {X -0.060,Y -143.034,Z 1277.172,A 0.000,B 0.000,C 90.000,E1 211.003} C_DIS
LIN {X 0.068,Y -141.658,Z 1277.152,A 0.000,B 0.000,C 90.000,E1 207.257} C_DIS
LIN {X -0.013,Y -139.447,Z 1277.115,A 0.000,B 0.000,C 90.000,E1 200.791} C_DIS
LIN {X 0.039,Y -139.180,Z 1277.105,A 0.000,B 0.000,C 90.000,E1 198.906} C_DIS
LIN {X 0.067,Y -138.321,Z 1277.053,A 0.000,B 0.000,C 90.000,E1 189.557} C_DIS
LIN {X -0.063,Y -139.465,Z 1277.007,A 0.000,B 0.000,C 90.000,E1 181.203} C_DIS
LIN {X 0.018,Y -141.028,Z 1276.975,A 0.000,B 0.000,C 90.000,E1 175.584} C_DIS
LIN {X -0.028,Y -142.394,Z 1276.960,A 0.000,B 0.000,C 90.000,E1 172.818} C_DIS
LIN {X 0.034,Y -144.625,Z 1276.934,A 0.000,B 0.000,C 90.000,E1 168.173} C_DIS
LIN {X -0.047,Y -147.821,Z 1276.909,A 0.000,B 0.000,C 90.000,E1 163.614} C_DIS
LIN {X 0.040,Y -150.512,Z 1276.889,A 0.000,B 0.000,C 90.000,E1 159.934} C_DIS
LIN {X 0.060,Y -153.972,Z 1276.869,A 0.000,B 0.000,C 90.000,E1 156.305} C_DIS
LIN {X -0.019,Y -157.384,Z 1276.849,A 0.000,B 0.000,C 90.000,E1 152.743} C_DIS
LIN {X -0.077,Y -161.587,Z 1276.829,A 0.000,B 0.000,C 90.000,E1 149.203} C_DIS
LIN {X -0.066,Y -165.784,Z 1276.809,A 0.000,B 0.000,C 90.000,E1 145.674} C_DIS
LIN {X -0.080,Y -170.746,Z 1276.790,A 0.000,B 0.000,C 90.000,E1 142.190} C_DIS
LIN {X 0.078,Y -175.618,Z 1276.771,A 0.000,B 0.000,C 90.000,E1 138.690} C_DIS
LIN {X -0.052,Y -181.234,Z 1276.752,A 0.000,B 0.000,C 90.000,E1 135.324} C_DIS
LIN {X 0.078,Y -186.702,Z 1276.733,A 0.000,B 0.000,C 90.000,E1 131.919} C_DIS
LIN {X 0.030,Y -191.302,Z 1276.719,A 0.000,B 0.000,C 90.000,E1 129.439} C_DIS
LIN {X -0.038,Y -197.131,Z 1276.701,A 0.000,B 0.000,C 90.000,E1 126.171} C_DIS
LIN {X 0.003,Y -199.908,Z 1276.693,A 0.000,B 0.000,C 90.000,E1 124.771} C_DIS
LIN {X 0.139,Y -309.392,Z 1276.693,A 0.000,B 0.000,C 90.000,E1 124.739} C_DIS
LIN {X -0.061,Y -313.733,Z 1276.693,A 0.000,B 0.000,C 90.000,E1 124.659} C_DIS
LIN {X -0.004,Y -315.759,Z 1276.692,A 0.000,B 0.000,C 90.000,E1 124.532} C_DIS
LIN {X -0.102,Y -319.621,Z 1276.690,A 0.000,B 0.000,C 90.000,E1 124.199} C_DIS
LIN {X 0.017,Y -323.132,Z 1276.687,A 0.000,B 0.000,C 90.000,E1 123.658} C_DIS
LIN {X -0.173,Y -324.649,Z 1276.685,A 0.000,B 0.000,C 90.000,E1 123.372} C_DIS
LIN {X 0.039,Y -337.637,Z 1276.666,A 0.000,B 0.000,C 90.000,E1 119.873} C_DIS
LIN {X -0.135,Y -349.687,Z 1276.651,A 0.000,B 0.000,C 90.000,E1 117.129} C_DIS
LIN {X 0.019,Y -363.205,Z 1276.635,A 0.000,B 0.000,C 90.000,E1 114.387} C_DIS
LIN {X 0.011,Y -376.548,Z 1276.622,A 0.000,B 0.000,C 90.000,E1 112.025} C_DIS
LIN {X 0.070,Y -391.236,Z 1276.609,A 0.000,B 0.000,C 90.000,E1 109.704} C_DIS
LIN {X -0.009,Y -407.373,Z 1276.597,A 0.000,B 0.000,C 90.000,E1 107.457} C_DIS
LIN {X 0.054,Y -425.072,Z 1276.585,A 0.000,B 0.000,C 90.000,E1 105.245} C_DIS
LIN {X -0.037,Y -444.397,Z 1276.573,A 0.000,B 0.000,C 90.000,E1 103.119} C_DIS
LIN {X -0.026,Y -464.563,Z 1276.562,A 0.000,B 0.000,C 90.000,E1 101.130} C_DIS
LIN {X -0.020,Y -474.848,Z 1276.557,A 0.000,B 0.000,C 90.000,E1 100.197} C_DIS
LIN {X 0.063,Y -477.120,Z 1276.555,A 0.000,B 0.000,C 90.000,E1 99.962} C_DIS
LIN {X 0.144,Y -478.837,Z 1276.554,A 0.000,B 0.000,C 90.000,E1 99.726} C_DIS
LIN {X -0.063,Y -480.290,Z 1276.553,A 0.000,B 0.000,C 90.000,E1 99.500} C_DIS
LIN {X -0.191,Y -481.371,Z 1276.551,A 0.000,B 0.000,C 90.000,E1 99.265} C_DIS
LIN {X -0.030,Y -482.638,Z 1276.549,A 0.000,B 0.000,C 90.000,E1 98.746} C_DIS
LIN {X 0.210,Y -482.885,Z 1276.546,A 0.000,B 0.000,C 90.000,E1 98.219} C_DIS
LIN {X -0.093,Y -482.154,Z 1276.543,A 0.000,B 0.000,C 90.000,E1 97.757} C_DIS
LIN {X 0.086,Y -480.326,Z 1276.540,A 0.000,B 0.000,C 90.000,E1 97.239} C_DIS
LIN {X -0.036,Y -478.892,Z 1276.539,A 0.000,B 0.000,C 90.000,E1 97.004} C_DIS
LIN {X 0.101,Y -457.063,Z 1276.522,A 0.000,B 0.000,C 90.000,E1 93.955} C_DIS
LIN {X 0.149,Y -438.416,Z 1276.506,A 0.000,B 0.000,C 90.000,E1 91.088} C_DIS
LIN {X 0.173,Y -420.242,Z 1276.488,A 0.000,B 0.000,C 90.000,E1 87.879} C_DIS
LIN {X 0.037,Y -410.095,Z 1276.478,A 0.000,B 0.000,C 90.000,E1 85.988} C_DIS
LIN {X 0.154,Y -400.022,Z 1276.467,A 0.000,B 0.000,C 90.000,E1 84.033} C_DIS
LIN {X 0.148,Y -389.727,Z 1276.456,A 0.000,B 0.000,C 90.000,E1 82.064} C_DIS
LIN {X -0.088,Y -380.747,Z 1276.447,A 0.000,B 0.000,C 90.000,E1 80.387} C_DIS
LIN {X 0.015,Y -373.004,Z 1276.438,A 0.000,B 0.000,C 90.000,E1 78.926} C_DIS
LIN {X -0.004,Y -365.014,Z 1276.430,A 0.000,B 0.000,C 90.000,E1 77.465} C_DIS
LIN {X -0.103,Y -355.144,Z 1276.420,A 0.000,B 0.000,C 90.000,E1 75.700} C_DIS
LIN {X 0.058,Y -343.591,Z 1276.409,A 0.000,B 0.000,C 90.000,E1 73.559} C_DIS
LIN {X 0.058,Y -332.166,Z 1276.397,A 0.000,B 0.000,C 90.000,E1 71.402} C_DIS
LIN {X -0.075,Y -317.999,Z 1276.381,A 0.000,B 0.000,C 90.000,E1 68.592} C_DIS
LIN {X -0.021,Y -301.965,Z 1276.361,A 0.000,B 0.000,C 90.000,E1 65.025} C_DIS
LIN {X 0.058,Y -291.536,Z 1276.347,A 0.000,B 0.000,C 90.000,E1 62.359} C_DIS
LIN {X -0.078,Y -279.050,Z 1276.326,A 0.000,B 0.000,C 90.000,E1 58.663} C_DIS
LIN {X 0.062,Y -268.930,Z 1276.307,A 0.000,B 0.000,C 90.000,E1 55.182} C_DIS
LIN {X -0.097,Y -259.615,Z 1276.287,A 0.000,B 0.000,C 90.000,E1 51.698} C_DIS
LIN {X -0.155,Y -252.516,Z 1276.271,A 0.000,B 0.000,C 90.000,E1 48.852} C_DIS
LIN {X 0.099,Y -244.014,Z 1276.251,A 0.000,B 0.000,C 90.000,E1 45.162} C_DIS
LIN {X -0.028,Y -237.659,Z 1276.235,A 0.000,B 0.000,C 90.000,E1 42.243} C_DIS
LIN {X 0.133,Y -230.266,Z 1276.214,A 0.000,B 0.000,C 90.000,E1 38.463} C_DIS
LIN {X 0.035,Y -223.627,Z 1276.193,A 0.000,B 0.000,C 90.000,E1 34.692} C_DIS
LIN {X 0.015,Y -218.857,Z 1276.176,A 0.000,B 0.000,C 90.000,E1 31.623} C_DIS
LIN {X 0.083,Y -213.435,Z 1276.154,A 0.000,B 0.000,C 90.000,E1 27.719} C_DIS
LIN {X -0.044,Y -208.679,Z 1276.132,A 0.000,B 0.000,C 90.000,E1 23.823} C_DIS
LIN {X 0.039,Y -203.831,Z 1276.106,A 0.000,B 0.000,C 90.000,E1 19.033} C_DIS
LIN {X -0.056,Y -199.875,Z 1276.079,A 0.000,B 0.000,C 90.000,E1 14.245} C_DIS
LIN {X -0.021,Y -196.555,Z 1276.048,A 0.000,B 0.000,C 90.000,E1 8.568} C_DIS
LIN {X -0.036,Y -194.565,Z 1275.997,A 0.000,B 0.000,C 90.000,E1 359.542} C_DIS
LIN {X -0.030,Y -196.785,Z 1275.952,A 0.000,B 0.000,C 90.000,E1 351.376} C_DIS
LIN {X -0.046,Y -200.480,Z 1275.921,A 0.000,B 0.000,C 90.000,E1 345.700} C_DIS
LIN {X -0.004,Y -204.760,Z 1275.894,A 0.000,B 0.000,C 90.000,E1 340.859} C_DIS
LIN {X 0.000,Y -209.118,Z 1275.871,A 0.000,B 0.000,C 90.000,E1 336.869} C_DIS
LIN {X -0.010,Y -214.179,Z 1275.850,A 0.000,B 0.000,C 90.000,E1 332.922} C_DIS
LIN {X 0.064,Y -219.949,Z 1275.828,A 0.000,B 0.000,C 90.000,E1 328.997} C_DIS
LIN {X -0.099,Y -226.537,Z 1275.806,A 0.000,B 0.000,C 90.000,E1 325.182} C_DIS
LIN {X 0.091,Y -234.038,Z 1275.785,A 0.000,B 0.000,C 90.000,E1 321.331} C_DIS
LIN {X -0.101,Y -242.390,Z 1275.765,A 0.000,B 0.000,C 90.000,E1 317.634} C_DIS
LIN {X -0.069,Y -251.907,Z 1275.744,A 0.000,B 0.000,C 90.000,E1 313.947} C_DIS
LIN {X 0.055,Y -259.503,Z 1275.730,A 0.000,B 0.000,C 90.000,E1 311.391} C_DIS
LIN {X 0.011,Y -268.244,Z 1275.716,A 0.000,B 0.000,C 90.000,E1 308.910} C_DIS
LIN {X 0.109,Y -276.834,Z 1275.704,A 0.000,B 0.000,C 90.000,E1 306.790} C_DIS
LIN {X 0.040,Y -286.435,Z 1275.693,A 0.000,B 0.000,C 90.000,E1 304.739} C_DIS
LIN {X -0.178,Y -298.977,Z 1275.680,A 0.000,B 0.000,C 90.000,E1 302.418} C_DIS
LIN {X 0.061,Y -309.001,Z 1275.671,A 0.000,B 0.000,C 90.000,E1 300.718} C_DIS
LIN {X 0.107,Y -317.909,Z 1275.663,A 0.000,B 0.000,C 90.000,E1 299.411} C_DIS
LIN {X 0.065,Y -339.947,Z 1275.648,A 0.000,B 0.000,C 90.000,E1 296.565} C_DIS
LIN {X -0.051,Y -357.992,Z 1275.636,A 0.000,B 0.000,C 90.000,E1 294.463} C_DIS
LIN {X 0.095,Y -370.962,Z 1275.628,A 0.000,B 0.000,C 90.000,E1 292.950} C_DIS
LIN {X -0.231,Y -383.738,Z 1275.620,A 0.000,B 0.000,C 90.000,E1 291.535} C_DIS
LIN {X -0.167,Y -398.546,Z 1275.610,A 0.000,B 0.000,C 90.000,E1 289.812} C_DIS
LIN {X 0.212,Y -415.967,Z 1275.599,A 0.000,B 0.000,C 90.000,E1 287.873} C_DIS
LIN {X 0.091,Y -425.792,Z 1275.593,A 0.000,B 0.000,C 90.000,E1 286.804} C_DIS
LIN {X -0.144,Y -432.712,Z 1275.589,A 0.000,B 0.000,C 90.000,E1 286.024} C_DIS
LIN {X 0.103,Y -439.148,Z 1275.584,A 0.000,B 0.000,C 90.000,E1 285.190} C_DIS
LIN {X -0.023,Y -444.912,Z 1275.580,A 0.000,B 0.000,C 90.000,E1 284.411} C_DIS
LIN {X 0.230,Y -449.997,Z 1275.576,A 0.000,B 0.000,C 90.000,E1 283.592} C_DIS
LIN {X 0.090,Y -454.452,Z 1275.571,A 0.000,B 0.000,C 90.000,E1 282.827} C_DIS
LIN {X -0.007,Y -458.240,Z 1275.567,A 0.000,B 0.000,C 90.000,E1 282.063} C_DIS
LIN {X -0.080,Y -461.317,Z 1275.563,A 0.000,B 0.000,C 90.000,E1 281.299} C_DIS
LIN {X -0.054,Y -463.009,Z 1275.560,A 0.000,B 0.000,C 90.000,E1 280.782} C_DIS
LIN {X 0.072,Y -464.392,Z 1275.557,A 0.000,B 0.000,C 90.000,E1 280.254} C_DIS
LIN {X 0.205,Y -465.461,Z 1275.554,A 0.000,B 0.000,C 90.000,E1 279.726} C_DIS
LIN {X -0.193,Y -466.203,Z 1275.551,A 0.000,B 0.000,C 90.000,E1 279.265} C_DIS
LIN {X -0.121,Y -466.539,Z 1275.548,A 0.000,B 0.000,C 90.000,E1 278.746} C_DIS
LIN {X 0.025,Y -466.532,Z 1275.546,A 0.000,B 0.000,C 90.000,E1 278.219} C_DIS
LIN {X 0.105,Y -466.064,Z 1275.543,A 0.000,B 0.000,C 90.000,E1 277.701} C_DIS
LIN {X 0.185,Y -465.132,Z 1275.540,A 0.000,B 0.000,C 90.000,E1 277.182} C_DIS
LIN {X -0.197,Y -463.754,Z 1275.537,A 0.000,B 0.000,C 90.000,E1 276.720} C_DIS
LIN {X -0.122,Y -461.975,Z 1275.534,A 0.000,B 0.000,C 90.000,E1 276.201} C_DIS
LIN {X 0.221,Y -458.622,Z 1275.530,A 0.000,B 0.000,C 90.000,E1 275.391} C_DIS
LIN {X 0.031,Y -454.518,Z 1275.526,A 0.000,B 0.000,C 90.000,E1 274.645} C_DIS
LIN {X 0.013,Y -450.964,Z 1275.523,A 0.000,B 0.000,C 90.000,E1 274.131} C_DIS
LIN {X 0.012,Y -446.350,Z 1275.520,A 0.000,B 0.000,C 90.000,E1 273.612} C_DIS
LIN {X 0.207,Y -443.664,Z 1275.519,A 0.000,B 0.000,C 90.000,E1 273.326} C_DIS
LIN {X 0.009,Y -437.551,Z 1275.516,A 0.000,B 0.000,C 90.000,E1 272.865} C_DIS
LIN {X -0.111,Y -431.073,Z 1275.514,A 0.000,B 0.000,C 90.000,E1 272.465} C_DIS
LIN {X -0.154,Y -424.174,Z 1275.512,A 0.000,B 0.000,C 90.000,E1 272.121} C_DIS
LIN {X 0.213,Y -417.284,Z 1275.510,A 0.000,B 0.000,C 90.000,E1 271.776} C_DIS
LIN {X 0.125,Y -406.410,Z 1275.508,A 0.000,B 0.000,C 90.000,E1 271.432} C_DIS
LIN {X -0.003,Y -399.190,Z 1275.507,A 0.000,B 0.000,C 90.000,E1 271.260} C_DIS
LIN {X 0.046,Y -387.747,Z 1275.506,A 0.000,B 0.000,C 90.000,E1 271.031} C_DIS
LIN {X 0.067,Y -378.953,Z 1275.505,A 0.000,B 0.000,C 90.000,E1 270.917} C_DIS
LIN {X -0.127,Y -367.915,Z 1275.505,A 0.000,B 0.000,C 90.000,E1 270.859} C_DIS
LIN {X 0.116,Y -363.451,Z 1275.505,A 0.000,B 0.000,C 90.000,E1 270.802} C_DIS
LIN {X 0.027,Y -181.499,Z 1275.505,A 0.000,B 0.000,C 90.000,E1 270.802} C_DIS
LIN {X 0.074,Y -181.516,Z 1275.499,A 0.000,B 0.000,C 90.000,E1 269.771} C_DIS
LIN {X 0.017,Y -180.906,Z 1275.474,A 0.000,B 0.000,C 90.000,E1 265.412} C_DIS
LIN {X 0.073,Y -180.713,Z 1275.470,A 0.000,B 0.000,C 90.000,E1 264.552} C_DIS
LIN {X -0.008,Y -178.799,Z 1275.442,A 0.000,B 0.000,C 90.000,E1 259.511} C_DIS
LIN {X 0.068,Y -175.845,Z 1275.413,A 0.000,B 0.000,C 90.000,E1 254.393} C_DIS
LIN {X 0.068,Y -172.036,Z 1275.385,A 0.000,B 0.000,C 90.000,E1 249.263} C_DIS
LIN {X 0.043,Y -171.466,Z 1275.380,A 0.000,B 0.000,C 90.000,E1 248.411} C_DIS
LIN {X 0.024,Y -167.698,Z 1275.356,A 0.000,B 0.000,C 90.000,E1 244.101} C_DIS
LIN {X 0.038,Y -166.383,Z 1275.347,A 0.000,B 0.000,C 90.000,E1 242.359} C_DIS
LIN {X 0.028,Y -163.111,Z 1275.327,A 0.000,B 0.000,C 90.000,E1 238.869} C_DIS
LIN {X 0.079,Y -161.059,Z 1275.313,A 0.000,B 0.000,C 90.000,E1 236.215} C_DIS
LIN {X -0.034,Y -157.794,Z 1275.293,A 0.000,B 0.000,C 90.000,E1 232.718} C_DIS
LIN {X 0.005,Y -155.830,Z 1275.278,A 0.000,B 0.000,C 90.000,E1 230.033} C_DIS
LIN {X -0.038,Y -152.080,Z 1275.253,A 0.000,B 0.000,C 90.000,E1 225.567} C_DIS
LIN {X -0.019,Y -150.331,Z 1275.238,A 0.000,B 0.000,C 90.000,E1 222.852} C_DIS
LIN {X 0.002,Y -147.071,Z 1275.213,A 0.000,B 0.000,C 90.000,E1 218.302} C_DIS
LIN {X -0.094,Y -145.646,Z 1275.198,A 0.000,B 0.000,C 90.000,E1 215.598} C_DIS
LIN {X -0.089,Y -143.028,Z 1275.172,A 0.000,B 0.000,C 90.000,E1 211.003} C_DIS
LIN {X 0.037,Y -141.654,Z 1275.151,A 0.000,B 0.000,C 90.000,E1 207.257} C_DIS
LIN {X -0.044,Y -139.445,Z 1275.115,A 0.000,B 0.000,C 90.000,E1 200.791} C_DIS
LIN {X 0.009,Y -139.179,Z 1275.105,A 0.000,B 0.000,C 90.000,E1 198.906} C_DIS
LIN {X 0.038,Y -138.320,Z 1275.053,A 0.000,B 0.000,C 90.000,E1 189.557} C_DIS
LIN {X 0.047,Y -139.467,Z 1275.006,A 0.000,B 0.000,C 90.000,E1 181.146} C_DIS
LIN {X -0.012,Y -141.033,Z 1274.975,A 0.000,B 0.000,C 90.000,E1 175.584} C_DIS
LIN {X -0.058,Y -142.400,Z 1274.960,A 0.000,B 0.000,C 90.000,E1 172.818} C_DIS
LIN {X 0.004,Y -144.632,Z 1274.934,A 0.000,B 0.000,C 90.000,E1 168.173} C_DIS
LIN {X 0.065,Y -147.828,Z 1274.909,A 0.000,B 0.000,C 90.000,E1 163.559} C_DIS
LIN {X 0.009,Y -150.521,Z 1274.889,A 0.000,B 0.000,C 90.000,E1 159.934} C_DIS
LIN {X 0.028,Y -153.984,Z 1274.868,A 0.000,B 0.000,C 90.000,E1 156.305} C_DIS
LIN {X -0.051,Y -157.396,Z 1274.849,A 0.000,B 0.000,C 90.000,E1 152.743} C_DIS
LIN {X 0.030,Y -161.602,Z 1274.829,A 0.000,B 0.000,C 90.000,E1 149.154} C_DIS
LIN {X -0.099,Y -165.799,Z 1274.809,A 0.000,B 0.000,C 90.000,E1 145.674} C_DIS
LIN {X 0.021,Y -170.763,Z 1274.790,A 0.000,B 0.000,C 90.000,E1 142.145} C_DIS
LIN {X 0.044,Y -175.635,Z 1274.771,A 0.000,B 0.000,C 90.000,E1 138.690} C_DIS
LIN {X -0.087,Y -181.250,Z 1274.752,A 0.000,B 0.000,C 90.000,E1 135.324} C_DIS
LIN {X 0.043,Y -186.722,Z 1274.733,A 0.000,B 0.000,C 90.000,E1 131.919} C_DIS
LIN {X -0.006,Y -191.320,Z 1274.719,A 0.000,B 0.000,C 90.000,E1 129.439} C_DIS
LIN {X -0.076,Y -197.152,Z 1274.701,A 0.000,B 0.000,C 90.000,E1 126.171} C_DIS
LIN {X 0.052,Y -199.946,Z 1274.693,A 0.000,B 0.000,C 90.000,E1 124.739} C_DIS
LIN {X 0.044,Y -309.605,Z 1274.693,A 0.000,B 0.000,C 90.000,E1 124.739} C_DIS
LIN {X -0.068,Y -310.992,Z 1274.693,A 0.000,B 0.000,C 90.000,E1 124.739} C_DIS
LIN {X -0.062,Y -315.709,Z 1274.692,A 0.000,B 0.000,C 90.000,E1 124.532} C_DIS
LIN {X 0.020,Y -318.883,Z 1274.690,A 0.000,B 0.000,C 90.000,E1 124.246} C_DIS
LIN {X -0.167,Y -322.546,Z 1274.688,A 0.000,B 0.000,C 90.000,E1 123.785} C_DIS
LIN {X 0.089,Y -324.202,Z 1274.686,A 0.000,B 0.000,C 90.000,E1 123.420} C_DIS
LIN {X -0.010,Y -326.599,Z 1274.682,A 0.000,B 0.000,C 90.000,E1 122.801} C_DIS
LIN {X -0.175,Y -337.245,Z 1274.667,A 0.000,B 0.000,C 90.000,E1 120.001} C_DIS
LIN {X -0.059,Y -349.248,Z 1274.651,A 0.000,B 0.000,C 90.000,E1 117.206} C_DIS
LIN {X 0.094,Y -362.717,Z 1274.636,A 0.000,B 0.000,C 90.000,E1 114.463} C_DIS
LIN {X 0.085,Y -376.012,Z 1274.623,A 0.000,B 0.000,C 90.000,E1 112.099} C_DIS
LIN {X -0.095,Y -390.649,Z 1274.610,A 0.000,B 0.000,C 90.000,E1 109.812} C_DIS
LIN {X 0.183,Y -406.730,Z 1274.597,A 0.000,B 0.000,C 90.000,E1 107.511} C_DIS
LIN {X 0.121,Y -424.369,Z 1274.585,A 0.000,B 0.000,C 90.000,E1 105.315} C_DIS
LIN {X 0.120,Y -443.641,Z 1274.573,A 0.000,B 0.000,C 90.000,E1 103.175} C_DIS
LIN {X 0.084,Y -463.786,Z 1274.562,A 0.000,B 0.000,C 90.000,E1 101.186} C_DIS
LIN {X 0.143,Y -476.475,Z 1274.556,A 0.000,B 0.000,C 90.000,E1 100.018} C_DIS
LIN {X 0.139,Y -478.317,Z 1274.554,A 0.000,B 0.000,C 90.000,E1 99.792} C_DIS
LIN {X 0.010,Y -479.867,Z 1274.553,A 0.000,B 0.000,C 90.000,E1 99.557} C_DIS
LIN {X -0.119,Y -481.026,Z 1274.552,A 0.000,B 0.000,C 90.000,E1 99.321} C_DIS
LIN {X 0.038,Y -482.417,Z 1274.549,A 0.000,B 0.000,C 90.000,E1 98.803} C_DIS
LIN {X -0.202,Y -482.774,Z 1274.546,A 0.000,B 0.000,C 90.000,E1 98.333} C_DIS
LIN {X -0.028,Y -482.155,Z 1274.543,A 0.000,B 0.000,C 90.000,E1 97.814} C_DIS
LIN {X 0.148,Y -480.464,Z 1274.541,A 0.000,B 0.000,C 90.000,E1 97.296} C_DIS
LIN {X -0.033,Y -479.119,Z 1274.539,A 0.000,B 0.000,C 90.000,E1 97.068} C_DIS
LIN {X 0.166,Y -457.327,Z 1274.522,A 0.000,B 0.000,C 90.000,E1 94.012} C_DIS
LIN {X 0.218,Y -438.620,Z 1274.506,A 0.000,B 0.000,C 90.000,E1 91.146} C_DIS
LIN {X -0.174,Y -420.398,Z 1274.489,A 0.000,B 0.000,C 90.000,E1 87.993} C_DIS
LIN {X -0.188,Y -408.832,Z 1274.477,A 0.000,B 0.000,C 90.000,E1 85.812} C_DIS
LIN {X -0.087,Y -398.750,Z 1274.466,A 0.000,B 0.000,C 90.000,E1 83.856} C_DIS
LIN {X -0.154,Y -388.432,Z 1274.455,A 0.000,B 0.000,C 90.000,E1 81.894} C_DIS
LIN {X 0.028,Y -379.429,Z 1274.445,A 0.000,B 0.000,C 90.000,E1 80.151} C_DIS
LIN {X 0.037,Y -370.056,Z 1274.436,A 0.000,B 0.000,C 90.000,E1 78.409} C_DIS
LIN {X 0.022,Y -360.334,Z 1274.426,A 0.000,B 0.000,C 90.000,E1 76.645} C_DIS
LIN {X -0.143,Y -348.789,Z 1274.414,A 0.000,B 0.000,C 90.000,E1 74.574} C_DIS
LIN {X -0.019,Y -337.305,Z 1274.402,A 0.000,B 0.000,C 90.000,E1 72.417} C_DIS
LIN {X 0.184,Y -322.915,Z 1274.387,A 0.000,B 0.000,C 90.000,E1 69.571} C_DIS
LIN {X 0.146,Y -306.426,Z 1274.367,A 0.000,B 0.000,C 90.000,E1 66.049} C_DIS
LIN {X -0.069,Y -294.267,Z 1274.351,A 0.000,B 0.000,C 90.000,E1 63.127} C_DIS
LIN {X 0.055,Y -283.619,Z 1274.334,A 0.000,B 0.000,C 90.000,E1 60.078} C_DIS
LIN {X 0.165,Y -272.983,Z 1274.315,A 0.000,B 0.000,C 90.000,E1 56.628} C_DIS
LIN {X -0.023,Y -263.300,Z 1274.295,A 0.000,B 0.000,C 90.000,E1 53.176} C_DIS
LIN {X -0.110,Y -256.057,Z 1274.280,A 0.000,B 0.000,C 90.000,E1 50.356} C_DIS
LIN {X -0.090,Y -249.044,Z 1274.264,A 0.000,B 0.000,C 90.000,E1 47.472} C_DIS
LIN {X 0.044,Y -240.801,Z 1274.243,A 0.000,B 0.000,C 90.000,E1 43.785} C_DIS
LIN {X -0.052,Y -233.081,Z 1274.223,A 0.000,B 0.000,C 90.000,E1 40.092} C_DIS
LIN {X 0.029,Y -226.133,Z 1274.202,A 0.000,B 0.000,C 90.000,E1 36.297} C_DIS
LIN {X 0.036,Y -219.873,Z 1274.180,A 0.000,B 0.000,C 90.000,E1 32.467} C_DIS
LIN {X -0.061,Y -214.252,Z 1274.159,A 0.000,B 0.000,C 90.000,E1 28.615} C_DIS
LIN {X 0.118,Y -209.310,Z 1274.137,A 0.000,B 0.000,C 90.000,E1 24.643} C_DIS
LIN {X -0.089,Y -204.256,Z 1274.111,A 0.000,B 0.000,C 90.000,E1 19.939} C_DIS
LIN {X -0.110,Y -200.117,Z 1274.084,A 0.000,B 0.000,C 90.000,E1 15.134} C_DIS
LIN {X -0.019,Y -196.577,Z 1274.052,A 0.000,B 0.000,C 90.000,E1 9.443} C_DIS
LIN {X 0.076,Y -194.293,Z 1274.007,A 0.000,B 0.000,C 90.000,E1 1.260} C_DIS
LIN {X -0.028,Y -196.209,Z 1273.957,A 0.000,B 0.000,C 90.000,E1 352.186} C_DIS
LIN {X 0.087,Y -199.735,Z 1273.925,A 0.000,B 0.000,C 90.000,E1 346.464} C_DIS
LIN {X 0.052,Y -203.901,Z 1273.898,A 0.000,B 0.000,C 90.000,E1 341.638} C_DIS
LIN {X -0.039,Y -208.130,Z 1273.876,A 0.000,B 0.000,C 90.000,E1 337.667} C_DIS
LIN {X 0.024,Y -213.082,Z 1273.854,A 0.000,B 0.000,C 90.000,E1 333.691} C_DIS
LIN {X -0.040,Y -218.734,Z 1273.832,A 0.000,B 0.000,C 90.000,E1 329.793} C_DIS
LIN {X -0.052,Y -225.134,Z 1273.811,A 0.000,B 0.000,C 90.000,E1 325.928} C_DIS
LIN {X -0.037,Y -232.480,Z 1273.789,A 0.000,B 0.000,C 90.000,E1 322.110} C_DIS
LIN {X 0.089,Y -240.622,Z 1273.769,A 0.000,B 0.000,C 90.000,E1 318.324} C_DIS
LIN {X -0.102,Y -249.863,Z 1273.748,A 0.000,B 0.000,C 90.000,E1 314.676} C_DIS
LIN {X -0.021,Y -258.336,Z 1273.732,A 0.000,B 0.000,C 90.000,E1 311.757} C_DIS
LIN {X -0.154,Y -265.602,Z 1273.720,A 0.000,B 0.000,C 90.000,E1 309.644} C_DIS
LIN {X -0.024,Y -272.363,Z 1273.710,A 0.000,B 0.000,C 90.000,E1 307.855} C_DIS
LIN {X 0.042,Y -281.467,Z 1273.699,A 0.000,B 0.000,C 90.000,E1 305.758} C_DIS
LIN {X 0.064,Y -291.605,Z 1273.687,A 0.000,B 0.000,C 90.000,E1 303.706} C_DIS
LIN {X -0.068,Y -300.841,Z 1273.678,A 0.000,B 0.000,C 90.000,E1 302.054} C_DIS
LIN {X 0.047,Y -311.067,Z 1273.669,A 0.000,B 0.000,C 90.000,E1 300.384} C_DIS
LIN {X 0.172,Y -322.605,Z 1273.660,A 0.000,B 0.000,C 90.000,E1 298.743} C_DIS
LIN {X -0.148,Y -344.974,Z 1273.644,A 0.000,B 0.000,C 90.000,E1 295.976} C_DIS
LIN {X 0.088,Y -360.546,Z 1273.634,A 0.000,B 0.000,C 90.000,E1 294.131} C_DIS
LIN {X -0.137,Y -376.089,Z 1273.624,A 0.000,B 0.000,C 90.000,E1 292.386} C_DIS
LIN {X -0.014,Y -388.693,Z 1273.616,A 0.000,B 0.000,C 90.000,E1 290.918} C_DIS
LIN {X 0.090,Y -408.612,Z 1273.604,A 0.000,B 0.000,C 90.000,E1 288.671} C_DIS
LIN {X 0.094,Y -418.756,Z 1273.598,A 0.000,B 0.000,C 90.000,E1 287.583} C_DIS
LIN {X -0.183,Y -426.092,Z 1273.593,A 0.000,B 0.000,C 90.000,E1 286.804} C_DIS
LIN {X -0.005,Y -433.003,Z 1273.589,A 0.000,B 0.000,C 90.000,E1 285.969} C_DIS
LIN {X -0.174,Y -439.403,Z 1273.584,A 0.000,B 0.000,C 90.000,E1 285.190} C_DIS
LIN {X 0.129,Y -445.135,Z 1273.580,A 0.000,B 0.000,C 90.000,E1 284.356} C_DIS
LIN {X -0.051,Y -450.241,Z 1273.575,A 0.000,B 0.000,C 90.000,E1 283.592} C_DIS
LIN {X 0.001,Y -453.295,Z 1273.573,A 0.000,B 0.000,C 90.000,E1 283.063} C_DIS
LIN {X -0.112,Y -457.234,Z 1273.568,A 0.000,B 0.000,C 90.000,E1 282.299} C_DIS
LIN {X -0.017,Y -459.453,Z 1273.565,A 0.000,B 0.000,C 90.000,E1 281.771} C_DIS
LIN {X 0.091,Y -461.426,Z 1273.563,A 0.000,B 0.000,C 90.000,E1 281.243} C_DIS
LIN {X 0.119,Y -463.128,Z 1273.560,A 0.000,B 0.000,C 90.000,E1 280.725} C_DIS
LIN {X -0.210,Y -464.458,Z 1273.557,A 0.000,B 0.000,C 90.000,E1 280.254} C_DIS
LIN {X -0.078,Y -465.528,Z 1273.554,A 0.000,B 0.000,C 90.000,E1 279.726} C_DIS
LIN {X -0.015,Y -466.231,Z 1273.551,A 0.000,B 0.000,C 90.000,E1 279.208} C_DIS
LIN {X 0.129,Y -466.608,Z 1273.548,A 0.000,B 0.000,C 90.000,E1 278.681} C_DIS
LIN {X 0.205,Y -466.548,Z 1273.546,A 0.000,B 0.000,C 90.000,E1 278.163} C_DIS
LIN {X -0.177,Y -466.092,Z 1273.543,A 0.000,B 0.000,C 90.000,E1 277.701} C_DIS
LIN {X -0.095,Y -465.180,Z 1273.540,A 0.000,B 0.000,C 90.000,E1 277.182} C_DIS
LIN {X -0.015,Y -463.810,Z 1273.537,A 0.000,B 0.000,C 90.000,E1 276.663} C_DIS
LIN {X 0.059,Y -462.049,Z 1273.534,A 0.000,B 0.000,C 90.000,E1 276.144} C_DIS
LIN {X -0.055,Y -458.715,Z 1273.530,A 0.000,B 0.000,C 90.000,E1 275.391} C_DIS
LIN {X -0.051,Y -456.097,Z 1273.527,A 0.000,B 0.000,C 90.000,E1 274.878} C_DIS
LIN {X 0.211,Y -454.635,Z 1273.526,A 0.000,B 0.000,C 90.000,E1 274.588} C_DIS
LIN {X 0.194,Y -451.088,Z 1273.523,A 0.000,B 0.000,C 90.000,E1 274.073} C_DIS
LIN {X -0.016,Y -448.936,Z 1273.521,A 0.000,B 0.000,C 90.000,E1 273.841} C_DIS
LIN {X -0.057,Y -443.745,Z 1273.518,A 0.000,B 0.000,C 90.000,E1 273.326} C_DIS
LIN {X 0.162,Y -440.663,Z 1273.517,A 0.000,B 0.000,C 90.000,E1 273.037} C_DIS
LIN {X 0.178,Y -437.652,Z 1273.516,A 0.000,B 0.000,C 90.000,E1 272.808} C_DIS
LIN {X 0.058,Y -431.082,Z 1273.513,A 0.000,B 0.000,C 90.000,E1 272.407} C_DIS
LIN {X 0.012,Y -424.172,Z 1273.511,A 0.000,B 0.000,C 90.000,E1 272.064} C_DIS
LIN {X -0.036,Y -417.141,Z 1273.510,A 0.000,B 0.000,C 90.000,E1 271.776} C_DIS
LIN {X -0.145,Y -409.884,Z 1273.508,A 0.000,B 0.000,C 90.000,E1 271.547} C_DIS
LIN {X 0.044,Y -402.802,Z 1273.507,A 0.000,B 0.000,C 90.000,E1 271.318} C_DIS
LIN {X 0.049,Y -395.438,Z 1273.506,A 0.000,B 0.000,C 90.000,E1 271.146} C_DIS
LIN {X -0.127,Y -387.787,Z 1273.506,A 0.000,B 0.000,C 90.000,E1 271.031} C_DIS
LIN {X -0.098,Y -378.889,Z 1273.505,A 0.000,B 0.000,C 90.000,E1 270.917} C_DIS
LIN {X 0.087,Y -367.847,Z 1273.505,A 0.000,B 0.000,C 90.000,E1 270.802} C_DIS
LIN {X -0.034,Y -361.696,Z 1273.504,A 0.000,B 0.000,C 90.000,E1 270.802} C_DIS
LIN {X -0.047,Y -181.505,Z 1273.504,A 0.000,B 0.000,C 90.000,E1 270.802} C_DIS
LIN {X 0.000,Y -181.510,Z 1273.499,A 0.000,B 0.000,C 90.000,E1 269.771} C_DIS
LIN {X -0.058,Y -180.906,Z 1273.474,A 0.000,B 0.000,C 90.000,E1 265.412} C_DIS
LIN {X 0.016,Y -180.702,Z 1273.470,A 0.000,B 0.000,C 90.000,E1 264.546} C_DIS
LIN {X 0.094,Y -178.787,Z 1273.442,A 0.000,B 0.000,C 90.000,E1 259.454} C_DIS
LIN {X -0.005,Y -175.832,Z 1273.413,A 0.000,B 0.000,C 90.000,E1 254.393} C_DIS
LIN {X -0.004,Y -172.022,Z 1273.385,A 0.000,B 0.000,C 90.000,E1 249.263} C_DIS
LIN {X -0.028,Y -171.446,Z 1273.380,A 0.000,B 0.000,C 90.000,E1 248.411} C_DIS
LIN {X 0.026,Y -167.681,Z 1273.356,A 0.000,B 0.000,C 90.000,E1 244.076} C_DIS
LIN {X -0.033,Y -166.358,Z 1273.346,A 0.000,B 0.000,C 90.000,E1 242.359} C_DIS
LIN {X -0.041,Y -163.091,Z 1273.327,A 0.000,B 0.000,C 90.000,E1 238.869} C_DIS
LIN {X 0.010,Y -161.034,Z 1273.312,A 0.000,B 0.000,C 90.000,E1 236.215} C_DIS
LIN {X -0.007,Y -157.773,Z 1273.293,A 0.000,B 0.000,C 90.000,E1 232.683} C_DIS
LIN {X 0.056,Y -155.811,Z 1273.278,A 0.000,B 0.000,C 90.000,E1 229.989} C_DIS
LIN {X 0.005,Y -152.063,Z 1273.253,A 0.000,B 0.000,C 90.000,E1 225.526} C_DIS
LIN {X -0.085,Y -150.312,Z 1273.238,A 0.000,B 0.000,C 90.000,E1 222.852} C_DIS
LIN {X 0.053,Y -147.056,Z 1273.213,A 0.000,B 0.000,C 90.000,E1 218.257} C_DIS
LIN {X 0.045,Y -145.633,Z 1273.197,A 0.000,B 0.000,C 90.000,E1 215.518} C_DIS
LIN {X 0.043,Y -143.016,Z 1273.172,A 0.000,B 0.000,C 90.000,E1 210.924} C_DIS
LIN {X -0.026,Y -141.643,Z 1273.151,A 0.000,B 0.000,C 90.000,E1 207.257} C_DIS
LIN {X 0.024,Y -139.440,Z 1273.115,A 0.000,B 0.000,C 90.000,E1 200.737} C_DIS
LIN {X -0.053,Y -139.173,Z 1273.105,A 0.000,B 0.000,C 90.000,E1 198.906} C_DIS
LIN {X -0.025,Y -138.318,Z 1273.053,A 0.000,B 0.000,C 90.000,E1 189.557} C_DIS
LIN {X -0.016,Y -139.472,Z 1273.006,A 0.000,B 0.000,C 90.000,E1 181.146} C_DIS
LIN {X 0.065,Y -141.044,Z 1272.975,A 0.000,B 0.000,C 90.000,E1 175.527} C_DIS
LIN {X 0.019,Y -142.414,Z 1272.960,A 0.000,B 0.000,C 90.000,E1 172.761} C_DIS
LIN {X -0.060,Y -144.648,Z 1272.934,A 0.000,B 0.000,C 90.000,E1 168.173} C_DIS
LIN {X -0.001,Y -147.844,Z 1272.909,A 0.000,B 0.000,C 90.000,E1 163.559} C_DIS
LIN {X -0.057,Y -150.543,Z 1272.888,A 0.000,B 0.000,C 90.000,E1 159.934} C_DIS
LIN {X -0.038,Y -154.009,Z 1272.868,A 0.000,B 0.000,C 90.000,E1 156.305} C_DIS
LIN {X 0.021,Y -157.422,Z 1272.848,A 0.000,B 0.000,C 90.000,E1 152.692} C_DIS
LIN {X 0.043,Y -161.635,Z 1272.829,A 0.000,B 0.000,C 90.000,E1 149.125} C_DIS
LIN {X 0.061,Y -165.831,Z 1272.809,A 0.000,B 0.000,C 90.000,E1 145.595} C_DIS
LIN {X 0.054,Y -170.802,Z 1272.790,A 0.000,B 0.000,C 90.000,E1 142.110} C_DIS
LIN {X -0.029,Y -175.671,Z 1272.771,A 0.000,B 0.000,C 90.000,E1 138.690} C_DIS
LIN {X 0.095,Y -181.284,Z 1272.751,A 0.000,B 0.000,C 90.000,E1 135.243} C_DIS
LIN {X -0.033,Y -186.763,Z 1272.733,A 0.000,B 0.000,C 90.000,E1 131.919} C_DIS
LIN {X 0.039,Y -191.357,Z 1272.719,A 0.000,B 0.000,C 90.000,E1 129.402} C_DIS
LIN {X -0.037,Y -197.195,Z 1272.701,A 0.000,B 0.000,C 90.000,E1 126.137} C_DIS
LIN {X 0.001,Y -199.976,Z 1272.693,A 0.000,B 0.000,C 90.000,E1 124.739} C_DIS
LIN {X -0.040,Y -309.485,Z 1272.693,A 0.000,B 0.000,C 90.000,E1 124.739} C_DIS
LIN {X 0.015,Y -313.806,Z 1272.692,A 0.000,B 0.000,C 90.000,E1 124.612} C_DIS
LIN {X 0.073,Y -315.831,Z 1272.692,A 0.000,B 0.000,C 90.000,E1 124.485} C_DIS
LIN {X 0.157,Y -319.694,Z 1272.690,A 0.000,B 0.000,C 90.000,E1 124.119} C_DIS
LIN {X 0.009,Y -323.205,Z 1272.687,A 0.000,B 0.000,C 90.000,E1 123.627} C_DIS
LIN {X 0.089,Y -324.721,Z 1272.685,A 0.000,B 0.000,C 90.000,E1 123.293} C_DIS
LIN {X -0.154,Y -337.727,Z 1272.666,A 0.000,B 0.000,C 90.000,E1 119.873} C_DIS
LIN {X -0.021,Y -349.791,Z 1272.650,A 0.000,B 0.000,C 90.000,E1 117.078} C_DIS
LIN {X 0.148,Y -363.328,Z 1272.635,A 0.000,B 0.000,C 90.000,E1 114.335} C_DIS
LIN {X -0.194,Y -376.687,Z 1272.622,A 0.000,B 0.000,C 90.000,E1 112.025} C_DIS
LIN {X -0.009,Y -391.394,Z 1272.609,A 0.000,B 0.000,C 90.000,E1 109.685} C_DIS
LIN {X 0.164,Y -407.551,Z 1272.597,A 0.000,B 0.000,C 90.000,E1 107.402} C_DIS
LIN {X -0.166,Y -425.271,Z 1272.585,A 0.000,B 0.000,C 90.000,E1 105.245} C_DIS
LIN {X 0.174,Y -444.615,Z 1272.573,A 0.000,B 0.000,C 90.000,E1 103.063} C_DIS
LIN {X -0.240,Y -464.788,Z 1272.562,A 0.000,B 0.000,C 90.000,E1 101.130} C_DIS
LIN {X -0.230,Y -475.073,Z 1272.557,A 0.000,B 0.000,C 90.000,E1 100.197} C_DIS
LIN {X -0.175,Y -477.247,Z 1272.555,A 0.000,B 0.000,C 90.000,E1 99.962} C_DIS
LIN {X -0.121,Y -478.894,Z 1272.554,A 0.000,B 0.000,C 90.000,E1 99.726} C_DIS
LIN {X 0.146,Y -480.265,Z 1272.553,A 0.000,B 0.000,C 90.000,E1 99.443} C_DIS
LIN {X 0.019,Y -481.283,Z 1272.551,A 0.000,B 0.000,C 90.000,E1 99.208} C_DIS
LIN {X 0.180,Y -482.445,Z 1272.548,A 0.000,B 0.000,C 90.000,E1 98.690} C_DIS
LIN {X -0.057,Y -482.600,Z 1272.546,A 0.000,B 0.000,C 90.000,E1 98.219} C_DIS
LIN {X 0.117,Y -481.770,Z 1272.543,A 0.000,B 0.000,C 90.000,E1 97.701} C_DIS
LIN {X -0.183,Y -479.822,Z 1272.540,A 0.000,B 0.000,C 90.000,E1 97.239} C_DIS
LIN {X 0.170,Y -478.307,Z 1272.539,A 0.000,B 0.000,C 90.000,E1 96.947} C_DIS
LIN {X -0.010,Y -461.763,Z 1272.526,A 0.000,B 0.000,C 90.000,E1 94.702} C_DIS
LIN {X -0.003,Y -444.386,Z 1272.512,A 0.000,B 0.000,C 90.000,E1 92.121} C_DIS
LIN {X 0.083,Y -431.532,Z 1272.500,A 0.000,B 0.000,C 90.000,E1 90.000} C_DIS
LIN {X 0.191,Y -415.272,Z 1272.484,A 0.000,B 0.000,C 90.000,E1 87.020} C_DIS
LIN {X 0.066,Y -403.780,Z 1272.471,A 0.000,B 0.000,C 90.000,E1 84.837} C_DIS
LIN {X 0.029,Y -395.057,Z 1272.462,A 0.000,B 0.000,C 90.000,E1 83.166} C_DIS
LIN {X -0.067,Y -384.688,Z 1272.451,A 0.000,B 0.000,C 90.000,E1 81.197} C_DIS
LIN {X 0.045,Y -375.537,Z 1272.441,A 0.000,B 0.000,C 90.000,E1 79.454} C_DIS
LIN {X 0.054,Y -366.028,Z 1272.432,A 0.000,B 0.000,C 90.000,E1 77.701} C_DIS
LIN {X -0.029,Y -356.198,Z 1272.422,A 0.000,B 0.000,C 90.000,E1 75.936} C_DIS
LIN {X 0.149,Y -344.680,Z 1272.410,A 0.000,B 0.000,C 90.000,E1 73.795} C_DIS
LIN {X 0.051,Y -331.622,Z 1272.396,A 0.000,B 0.000,C 90.000,E1 71.348} C_DIS
LIN {X -0.047,Y -319.071,Z 1272.382,A 0.000,B 0.000,C 90.000,E1 68.847} C_DIS
LIN {X 0.039,Y -302.964,Z 1272.363,A 0.000,B 0.000,C 90.000,E1 65.281} C_DIS
LIN {X 0.141,Y -292.448,Z 1272.348,A 0.000,B 0.000,C 90.000,E1 62.615} C_DIS
LIN {X 0.028,Y -279.753,Z 1272.327,A 0.000,B 0.000,C 90.000,E1 58.918} C_DIS
LIN {X 0.113,Y -268.469,Z 1272.306,A 0.000,B 0.000,C 90.000,E1 55.102} C_DIS
LIN {X -0.059,Y -259.077,Z 1272.287,A 0.000,B 0.000,C 90.000,E1 51.618} C_DIS
LIN {X -0.129,Y -251.973,Z 1272.271,A 0.000,B 0.000,C 90.000,E1 48.771} C_DIS
LIN {X 0.107,Y -243.461,Z 1272.251,A 0.000,B 0.000,C 90.000,E1 45.081} C_DIS
LIN {X -0.033,Y -237.135,Z 1272.234,A 0.000,B 0.000,C 90.000,E1 42.162} C_DIS
LIN {X 0.110,Y -229.693,Z 1272.213,A 0.000,B 0.000,C 90.000,E1 38.382} C_DIS
LIN {X -0.010,Y -222.965,Z 1272.192,A 0.000,B 0.000,C 90.000,E1 34.612} C_DIS
LIN {X 0.034,Y -216.975,Z 1272.171,A 0.000,B 0.000,C 90.000,E1 30.747} C_DIS
LIN {X -0.064,Y -211.590,Z 1272.149,A 0.000,B 0.000,C 90.000,E1 26.873} C_DIS
LIN {X 0.046,Y -206.922,Z 1272.127,A 0.000,B 0.000,C 90.000,E1 22.898} C_DIS
LIN {X -0.006,Y -202.190,Z 1272.101,A 0.000,B 0.000,C 90.000,E1 18.127} C_DIS
LIN {X -0.022,Y -198.432,Z 1272.074,A 0.000,B 0.000,C 90.000,E1 13.300} C_DIS
LIN {X 0.074,Y -195.388,Z 1272.042,A 0.000,B 0.000,C 90.000,E1 7.587} C_DIS
LIN {X -0.059,Y -196.433,Z 1271.952,A 0.000,B 0.000,C 90.000,E1 351.376} C_DIS
LIN {X 0.067,Y -199.611,Z 1271.925,A 0.000,B 0.000,C 90.000,E1 346.464} C_DIS
LIN {X 0.026,Y -203.805,Z 1271.898,A 0.000,B 0.000,C 90.000,E1 341.638} C_DIS
LIN {X 0.023,Y -208.993,Z 1271.871,A 0.000,B 0.000,C 90.000,E1 336.847} C_DIS
LIN {X 0.116,Y -214.102,Z 1271.849,A 0.000,B 0.000,C 90.000,E1 332.871} C_DIS
LIN {X -0.004,Y -219.907,Z 1271.828,A 0.000,B 0.000,C 90.000,E1 328.997} C_DIS
LIN {X 0.016,Y -226.536,Z 1271.806,A 0.000,B 0.000,C 90.000,E1 325.135} C_DIS
LIN {X 0.017,Y -234.020,Z 1271.785,A 0.000,B 0.000,C 90.000,E1 321.331} C_DIS
LIN {X -0.014,Y -242.360,Z 1271.764,A 0.000,B 0.000,C 90.000,E1 317.595} C_DIS
LIN {X -0.149,Y -251.842,Z 1271.744,A 0.000,B 0.000,C 90.000,E1 313.947} C_DIS
LIN {X -0.029,Y -259.454,Z 1271.730,A 0.000,B 0.000,C 90.000,E1 311.391} C_DIS
LIN {X -0.077,Y -268.169,Z 1271.716,A 0.000,B 0.000,C 90.000,E1 308.910} C_DIS
LIN {X 0.017,Y -276.747,Z 1271.704,A 0.000,B 0.000,C 90.000,E1 306.790} C_DIS
LIN {X -0.057,Y -286.360,Z 1271.693,A 0.000,B 0.000,C 90.000,E1 304.739} C_DIS
LIN {X 0.130,Y -296.997,Z 1271.682,A 0.000,B 0.000,C 90.000,E1 302.673} C_DIS
LIN {X -0.074,Y -306.779,Z 1271.672,A 0.000,B 0.000,C 90.000,E1 301.052} C_DIS
LIN {X -0.076,Y -315.451,Z 1271.665,A 0.000,B 0.000,C 90.000,E1 299.745} C_DIS
LIN {X -0.054,Y -337.312,Z 1271.649,A 0.000,B 0.000,C 90.000,E1 296.873} C_DIS
LIN {X 0.136,Y -358.089,Z 1271.636,A 0.000,B 0.000,C 90.000,E1 294.387} C_DIS
LIN {X -0.087,Y -370.935,Z 1271.627,A 0.000,B 0.000,C 90.000,E1 292.950} C_DIS
LIN {X 0.079,Y -383.771,Z 1271.619,A 0.000,B 0.000,C 90.000,E1 291.461} C_DIS
LIN {X 0.005,Y -398.695,Z 1271.610,A 0.000,B 0.000,C 90.000,E1 289.758} C_DIS
LIN {X -0.166,Y -416.390,Z 1271.599,A 0.000,B 0.000,C 90.000,E1 287.873} C_DIS
LIN {X 0.117,Y -426.201,Z 1271.593,A 0.000,B 0.000,C 90.000,E1 286.749} C_DIS
LIN {X -0.113,Y -433.104,Z 1271.589,A 0.000,B 0.000,C 90.000,E1 285.969} C_DIS
LIN {X 0.141,Y -439.494,Z 1271.584,A 0.000,B 0.000,C 90.000,E1 285.134} C_DIS
LIN {X 0.020,Y -445.250,Z 1271.580,A 0.000,B 0.000,C 90.000,E1 284.356} C_DIS
LIN {X -0.160,Y -450.322,Z 1271.575,A 0.000,B 0.000,C 90.000,E1 283.592} C_DIS
LIN {X 0.143,Y -454.727,Z 1271.571,A 0.000,B 0.000,C 90.000,E1 282.771} C_DIS
LIN {X -0.223,Y -457.271,Z 1271.568,A 0.000,B 0.000,C 90.000,E1 282.299} C_DIS
LIN {X -0.127,Y -459.502,Z 1271.565,A 0.000,B 0.000,C 90.000,E1 281.771} C_DIS
LIN {X -0.019,Y -461.451,Z 1271.563,A 0.000,B 0.000,C 90.000,E1 281.243} C_DIS
LIN {X 0.094,Y -463.120,Z 1271.560,A 0.000,B 0.000,C 90.000,E1 280.715} C_DIS
LIN {X 0.136,Y -464.486,Z 1271.557,A 0.000,B 0.000,C 90.000,E1 280.197} C_DIS
LIN {X -0.188,Y -465.547,Z 1271.554,A 0.000,B 0.000,C 90.000,E1 279.726} C_DIS
LIN {X -0.126,Y -466.297,Z 1271.551,A 0.000,B 0.000,C 90.000,E1 279.208} C_DIS
LIN {X 0.018,Y -466.634,Z 1271.548,A 0.000,B 0.000,C 90.000,E1 278.681} C_DIS
LIN {X 0.094,Y -466.607,Z 1271.545,A 0.000,B 0.000,C 90.000,E1 278.163} C_DIS
LIN {X 0.175,Y -466.166,Z 1271.543,A 0.000,B 0.000,C 90.000,E1 277.644} C_DIS
LIN {X -0.205,Y -465.280,Z 1271.540,A 0.000,B 0.000,C 90.000,E1 277.182} C_DIS
LIN {X -0.124,Y -463.956,Z 1271.537,A 0.000,B 0.000,C 90.000,E1 276.663} C_DIS
LIN {X -0.049,Y -462.190,Z 1271.534,A 0.000,B 0.000,C 90.000,E1 276.144} C_DIS
LIN {X -0.161,Y -458.910,Z 1271.530,A 0.000,B 0.000,C 90.000,E1 275.391} C_DIS
LIN {X -0.155,Y -456.332,Z 1271.527,A 0.000,B 0.000,C 90.000,E1 274.878} C_DIS
LIN {X -0.126,Y -453.237,Z 1271.524,A 0.000,B 0.000,C 90.000,E1 274.359} C_DIS
LIN {X -0.116,Y -449.236,Z 1271.521,A 0.000,B 0.000,C 90.000,E1 273.841} C_DIS
LIN {X -0.155,Y -444.097,Z 1271.518,A 0.000,B 0.000,C 90.000,E1 273.326} C_DIS
LIN {X 0.078,Y -438.041,Z 1271.516,A 0.000,B 0.000,C 90.000,E1 272.808} C_DIS
LIN {X 0.091,Y -434.696,Z 1271.514,A 0.000,B 0.000,C 90.000,E1 272.579} C_DIS
LIN {X 0.199,Y -427.767,Z 1271.512,A 0.000,B 0.000,C 90.000,E1 272.178} C_DIS
LIN {X -0.040,Y -420.817,Z 1271.510,A 0.000,B 0.000,C 90.000,E1 271.892} C_DIS
LIN {X 0.107,Y -413.636,Z 1271.509,A 0.000,B 0.000,C 90.000,E1 271.604} C_DIS
LIN {X -0.088,Y -403.161,Z 1271.507,A 0.000,B 0.000,C 90.000,E1 271.318} C_DIS
LIN {X 0.185,Y -391.933,Z 1271.506,A 0.000,B 0.000,C 90.000,E1 271.031} C_DIS
LIN {X 0.078,Y -383.390,Z 1271.505,A 0.000,B 0.000,C 90.000,E1 270.917} C_DIS
LIN {X -0.185,Y -373.292,Z 1271.505,A 0.000,B 0.000,C 90.000,E1 270.859} C_DIS
LIN {X -0.171,Y -361.512,Z 1271.504,A 0.000,B 0.000,C 90.000,E1 270.802} C_DIS
LIN {X 0.067,Y -181.510,Z 1271.504,A 0.000,B 0.000,C 90.000,E1 270.745} C_DIS
LIN {X -0.068,Y -181.505,Z 1271.499,A 0.000,B 0.000,C 90.000,E1 269.771} C_DIS
LIN {X 0.055,Y -180.907,Z 1271.474,A 0.000,B 0.000,C 90.000,E1 265.355} C_DIS
LIN {X -0.050,Y -180.691,Z 1271.470,A 0.000,B 0.000,C 90.000,E1 264.546} C_DIS
LIN {X 0.028,Y -178.775,Z 1271.441,A 0.000,B 0.000,C 90.000,E1 259.454} C_DIS
LIN {X -0.070,Y -175.821,Z 1271.413,A 0.000,B 0.000,C 90.000,E1 254.393} C_DIS
LIN {X -0.068,Y -172.009,Z 1271.385,A 0.000,B 0.000,C 90.000,E1 249.263} C_DIS
LIN {X -0.093,Y -171.427,Z 1271.380,A 0.000,B 0.000,C 90.000,E1 248.411} C_DIS
LIN {X -0.037,Y -167.664,Z 1271.356,A 0.000,B 0.000,C 90.000,E1 244.076} C_DIS
LIN {X -0.097,Y -166.335,Z 1271.346,A 0.000,B 0.000,C 90.000,E1 242.359} C_DIS
LIN {X 0.036,Y -163.073,Z 1271.327,A 0.000,B 0.000,C 90.000,E1 238.820} C_DIS
LIN {X -0.053,Y -161.012,Z 1271.312,A 0.000,B 0.000,C 90.000,E1 236.215} C_DIS
LIN {X 0.058,Y -157.756,Z 1271.293,A 0.000,B 0.000,C 90.000,E1 232.637} C_DIS
LIN {X -0.004,Y -155.793,Z 1271.278,A 0.000,B 0.000,C 90.000,E1 229.989} C_DIS
LIN {X 0.050,Y -152.047,Z 1271.253,A 0.000,B 0.000,C 90.000,E1 225.486} C_DIS
LIN {X 0.068,Y -150.296,Z 1271.238,A 0.000,B 0.000,C 90.000,E1 222.771} C_DIS
LIN {X -0.007,Y -147.043,Z 1271.213,A 0.000,B 0.000,C 90.000,E1 218.257} C_DIS
LIN {X -0.014,Y -145.622,Z 1271.197,A 0.000,B 0.000,C 90.000,E1 215.518} C_DIS
LIN {X -0.015,Y -143.006,Z 1271.172,A 0.000,B 0.000,C 90.000,E1 210.924} C_DIS
LIN {X 0.043,Y -141.632,Z 1271.151,A 0.000,B 0.000,C 90.000,E1 207.206} C_DIS
LIN {X -0.033,Y -139.436,Z 1271.115,A 0.000,B 0.000,C 90.000,E1 200.737} C_DIS
LIN {X 0.021,Y -139.168,Z 1271.105,A 0.000,B 0.000,C 90.000,E1 198.852} C_DIS
LIN {X 0.055,Y -138.317,Z 1271.053,A 0.000,B 0.000,C 90.000,E1 189.500} C_DIS
LIN {X 0.066,Y -139.474,Z 1271.006,A 0.000,B 0.000,C 90.000,E1 181.088} C_DIS
LIN {X 0.008,Y -141.054,Z 1270.975,A 0.000,B 0.000,C 90.000,E1 175.527} C_DIS
LIN {X -0.039,Y -142.426,Z 1270.960,A 0.000,B 0.000,C 90.000,E1 172.761} C_DIS
LIN {X 0.023,Y -144.662,Z 1270.934,A 0.000,B 0.000,C 90.000,E1 168.117} C_DIS
LIN {X 0.006,Y -147.245,Z 1270.914,A 0.000,B 0.000,C 90.000,E1 164.448} C_DIS
LIN {X 0.024,Y -150.562,Z 1270.888,A 0.000,B 0.000,C 90.000,E1 159.880} C_DIS
LIN {X -0.037,Y -154.031,Z 1270.868,A 0.000,B 0.000,C 90.000,E1 156.282} C_DIS
LIN {X 0.031,Y -157.446,Z 1270.848,A 0.000,B 0.000,C 90.000,E1 152.666} C_DIS
LIN {X -0.019,Y -161.664,Z 1270.828,A 0.000,B 0.000,C 90.000,E1 149.125} C_DIS
LIN {X -0.002,Y -165.858,Z 1270.809,A 0.000,B 0.000,C 90.000,E1 145.595} C_DIS
LIN {X -0.011,Y -170.835,Z 1270.789,A 0.000,B 0.000,C 90.000,E1 142.110} C_DIS
LIN {X 0.036,Y -175.704,Z 1270.770,A 0.000,B 0.000,C 90.000,E1 138.647} C_DIS
LIN {X 0.028,Y -181.316,Z 1270.751,A 0.000,B 0.000,C 90.000,E1 135.243} C_DIS
LIN {X -0.102,Y -186.800,Z 1270.733,A 0.000,B 0.000,C 90.000,E1 131.919} C_DIS
LIN {X -0.031,Y -191.391,Z 1270.719,A 0.000,B 0.000,C 90.000,E1 129.402} C_DIS
LIN {X 0.052,Y -197.236,Z 1270.701,A 0.000,B 0.000,C 90.000,E1 126.091} C_DIS
LIN {X -0.070,Y -200.019,Z 1270.693,A 0.000,B 0.000,C 90.000,E1 124.739} C_DIS
LIN {X 0.105,Y -309.962,Z 1270.693,A 0.000,B 0.000,C 90.000,E1 124.692} C_DIS
LIN {X -0.039,Y -315.928,Z 1270.692,A 0.000,B 0.000,C 90.000,E1 124.485} C_DIS
LIN {X -0.071,Y -318.796,Z 1270.690,A 0.000,B 0.000,C 90.000,E1 124.246} C_DIS
LIN {X 0.192,Y -322.516,Z 1270.688,A 0.000,B 0.000,C 90.000,E1 123.706} C_DIS
LIN {X 0.000,Y -324.195,Z 1270.686,A 0.000,B 0.000,C 90.000,E1 123.420} C_DIS
LIN {X 0.175,Y -326.612,Z 1270.682,A 0.000,B 0.000,C 90.000,E1 122.752} C_DIS
LIN {X 0.025,Y -337.265,Z 1270.666,A 0.000,B 0.000,C 90.000,E1 119.951} C_DIS
LIN {X 0.007,Y -349.275,Z 1270.651,A 0.000,B 0.000,C 90.000,E1 117.180} C_DIS
LIN {X -0.004,Y -362.752,Z 1270.636,A 0.000,B 0.000,C 90.000,E1 114.463} C_DIS
LIN {X 0.126,Y -376.054,Z 1270.623,A 0.000,B 0.000,C 90.000,E1 112.078} C_DIS
LIN {X 0.170,Y -390.700,Z 1270.610,A 0.000,B 0.000,C 90.000,E1 109.758} C_DIS
LIN {X 0.076,Y -406.790,Z 1270.597,A 0.000,B 0.000,C 90.000,E1 107.511} C_DIS
LIN {X 0.013,Y -424.440,Z 1270.585,A 0.000,B 0.000,C 90.000,E1 105.315} C_DIS
LIN {X 0.010,Y -443.721,Z 1270.573,A 0.000,B 0.000,C 90.000,E1 103.175} C_DIS
LIN {X -0.023,Y -463.869,Z 1270.562,A 0.000,B 0.000,C 90.000,E1 101.186} C_DIS
LIN {X -0.039,Y -474.147,Z 1270.557,A 0.000,B 0.000,C 90.000,E1 100.254} C_DIS
LIN {X 0.038,Y -476.486,Z 1270.556,A 0.000,B 0.000,C 90.000,E1 100.018} C_DIS
LIN {X 0.033,Y -478.258,Z 1270.554,A 0.000,B 0.000,C 90.000,E1 99.792} C_DIS
LIN {X -0.095,Y -479.753,Z 1270.553,A 0.000,B 0.000,C 90.000,E1 99.557} C_DIS
LIN {X -0.225,Y -480.870,Z 1270.552,A 0.000,B 0.000,C 90.000,E1 99.321} C_DIS
LIN {X -0.069,Y -482.193,Z 1270.549,A 0.000,B 0.000,C 90.000,E1 98.803} C_DIS
LIN {X 0.167,Y -482.491,Z 1270.546,A 0.000,B 0.000,C 90.000,E1 98.276} C_DIS
LIN {X -0.138,Y -481.813,Z 1270.543,A 0.000,B 0.000,C 90.000,E1 97.814} C_DIS
LIN {X 0.038,Y -480.049,Z 1270.541,A 0.000,B 0.000,C 90.000,E1 97.296} C_DIS
LIN {X -0.144,Y -478.658,Z 1270.539,A 0.000,B 0.000,C 90.000,E1 97.068} C_DIS
LIN {X -0.222,Y -458.614,Z 1270.524,A 0.000,B 0.000,C 90.000,E1 94.302} C_DIS
LIN {X -0.181,Y -436.507,Z 1270.505,A 0.000,B 0.000,C 90.000,E1 90.917} C_DIS
LIN {X -0.099,Y -416.984,Z 1270.486,A 0.000,B 0.000,C 90.000,E1 87.421} C_DIS
LIN {X -0.203,Y -405.504,Z 1270.473,A 0.000,B 0.000,C 90.000,E1 85.241} C_DIS
LIN {X -0.208,Y -396.812,Z 1270.464,A 0.000,B 0.000,C 90.000,E1 83.571} C_DIS
LIN {X 0.113,Y -386.458,Z 1270.453,A 0.000,B 0.000,C 90.000,E1 81.546} C_DIS
LIN {X -0.118,Y -377.401,Z 1270.444,A 0.000,B 0.000,C 90.000,E1 79.859} C_DIS
LIN {X -0.066,Y -367.976,Z 1270.434,A 0.000,B 0.000,C 90.000,E1 78.105} C_DIS
LIN {X -0.191,Y -358.207,Z 1270.424,A 0.000,B 0.000,C 90.000,E1 76.353} C_DIS
LIN {X 0.037,Y -346.706,Z 1270.412,A 0.000,B 0.000,C 90.000,E1 74.212} C_DIS
LIN {X -0.004,Y -333.606,Z 1270.399,A 0.000,B 0.000,C 90.000,E1 71.764} C_DIS
LIN {X -0.047,Y -321.001,Z 1270.385,A 0.000,B 0.000,C 90.000,E1 69.263} C_DIS
LIN {X -0.140,Y -304.711,Z 1270.365,A 0.000,B 0.000,C 90.000,E1 65.741} C_DIS
LIN {X 0.004,Y -294.032,Z 1270.350,A 0.000,B 0.000,C 90.000,E1 63.076} C_DIS
LIN {X 0.008,Y -283.345,Z 1270.334,A 0.000,B 0.000,C 90.000,E1 60.049} C_DIS
LIN {X -0.033,Y -272.612,Z 1270.315,A 0.000,B 0.000,C 90.000,E1 56.628} C_DIS
LIN {X -0.015,Y -262.833,Z 1270.295,A 0.000,B 0.000,C 90.000,E1 53.130} C_DIS
LIN {X 0.042,Y -255.572,Z 1270.279,A 0.000,B 0.000,C 90.000,E1 50.275} C_DIS
LIN {X 0.046,Y -248.546,Z 1270.263,A 0.000,B 0.000,C 90.000,E1 47.391} C_DIS
LIN {X -0.005,Y -240.295,Z 1270.243,A 0.000,B 0.000,C 90.000,E1 43.743} C_DIS
LIN {X -0.045,Y -234.070,Z 1270.227,A 0.000,B 0.000,C 90.000,E1 40.782} C_DIS
LIN {X 0.030,Y -226.881,Z 1270.206,A 0.000,B 0.000,C 90.000,E1 36.996} C_DIS
LIN {X 0.060,Y -220.385,Z 1270.184,A 0.000,B 0.000,C 90.000,E1 33.166} C_DIS
LIN {X 0.092,Y -214.533,Z 1270.163,A 0.000,B 0.000,C 90.000,E1 29.283} C_DIS
LIN {X -0.092,Y -209.400,Z 1270.141,A 0.000,B 0.000,C 90.000,E1 25.412} C_DIS
LIN {X 0.054,Y -204.950,Z 1270.119,A 0.000,B 0.000,C 90.000,E1 21.408} C_DIS
LIN {X -0.016,Y -200.502,Z 1270.092,A 0.000,B 0.000,C 90.000,E1 16.622} C_DIS
LIN {X 0.021,Y -196.596,Z 1270.061,A 0.000,B 0.000,C 90.000,E1 10.950} C_DIS
LIN {X 0.060,Y -194.061,Z 1270.025,A 0.000,B 0.000,C 90.000,E1 4.416} C_DIS
LIN {X -0.033,Y -195.449,Z 1269.961,A 0.000,B 0.000,C 90.000,E1 352.996} C_DIS
LIN {X 0.010,Y -198.844,Z 1269.929,A 0.000,B 0.000,C 90.000,E1 347.285} C_DIS
LIN {X 0.084,Y -202.937,Z 1269.902,A 0.000,B 0.000,C 90.000,E1 342.417} C_DIS
LIN {X -0.099,Y -207.980,Z 1269.876,A 0.000,B 0.000,C 90.000,E1 337.667} C_DIS
LIN {X -0.042,Y -212.994,Z 1269.854,A 0.000,B 0.000,C 90.000,E1 333.691} C_DIS
LIN {X 0.079,Y -218.686,Z 1269.832,A 0.000,B 0.000,C 90.000,E1 329.744} C_DIS
LIN {X 0.061,Y -225.110,Z 1269.811,A 0.000,B 0.000,C 90.000,E1 325.881} C_DIS
LIN {X 0.070,Y -232.433,Z 1269.789,A 0.000,B 0.000,C 90.000,E1 322.065} C_DIS
LIN {X 0.009,Y -240.592,Z 1269.768,A 0.000,B 0.000,C 90.000,E1 318.324} C_DIS
LIN {X -0.011,Y -249.813,Z 1269.748,A 0.000,B 0.000,C 90.000,E1 314.636} C_DIS
LIN {X -0.110,Y -258.273,Z 1269.732,A 0.000,B 0.000,C 90.000,E1 311.757} C_DIS
LIN {X -0.018,Y -266.802,Z 1269.718,A 0.000,B 0.000,C 90.000,E1 309.241} C_DIS
LIN {X -0.122,Y -275.189,Z 1269.706,A 0.000,B 0.000,C 90.000,E1 307.156} C_DIS
LIN {X 0.169,Y -284.639,Z 1269.695,A 0.000,B 0.000,C 90.000,E1 305.025} C_DIS
LIN {X -0.077,Y -295.091,Z 1269.683,A 0.000,B 0.000,C 90.000,E1 303.038} C_DIS
LIN {X 0.104,Y -304.644,Z 1269.674,A 0.000,B 0.000,C 90.000,E1 301.337} C_DIS
LIN {X -0.138,Y -315.356,Z 1269.665,A 0.000,B 0.000,C 90.000,E1 299.745} C_DIS
LIN {X -0.123,Y -337.240,Z 1269.649,A 0.000,B 0.000,C 90.000,E1 296.873} C_DIS
LIN {X 0.150,Y -357.901,Z 1269.636,A 0.000,B 0.000,C 90.000,E1 294.387} C_DIS
LIN {X -0.148,Y -370.859,Z 1269.627,A 0.000,B 0.000,C 90.000,E1 292.950} C_DIS
LIN {X 0.102,Y -383.623,Z 1269.619,A 0.000,B 0.000,C 90.000,E1 291.461} C_DIS
LIN {X 0.109,Y -398.499,Z 1269.610,A 0.000,B 0.000,C 90.000,E1 289.758} C_DIS
LIN {X -0.029,Y -416.201,Z 1269.599,A 0.000,B 0.000,C 90.000,E1 287.873} C_DIS
LIN {X 0.121,Y -423.618,Z 1269.595,A 0.000,B 0.000,C 90.000,E1 287.040} C_DIS
LIN {X -0.126,Y -430.668,Z 1269.590,A 0.000,B 0.000,C 90.000,E1 286.260} C_DIS
LIN {X 0.095,Y -437.263,Z 1269.586,A 0.000,B 0.000,C 90.000,E1 285.426} C_DIS
LIN {X -0.042,Y -443.230,Z 1269.581,A 0.000,B 0.000,C 90.000,E1 284.647} C_DIS
LIN {X 0.188,Y -448.596,Z 1269.577,A 0.000,B 0.000,C 90.000,E1 283.828} C_DIS
LIN {X 0.041,Y -453.225,Z 1269.573,A 0.000,B 0.000,C 90.000,E1 283.063} C_DIS
LIN {X -0.072,Y -457.171,Z 1269.568,A 0.000,B 0.000,C 90.000,E1 282.299} C_DIS
LIN {X 0.023,Y -459.397,Z 1269.565,A 0.000,B 0.000,C 90.000,E1 281.771} C_DIS
LIN {X 0.131,Y -461.341,Z 1269.563,A 0.000,B 0.000,C 90.000,E1 281.243} C_DIS
END
